(* Logix 5000 project; controller P1 vendor 1 type 14 code 92 rev 20.55; software revision 20.01 *)

TASK MainTask (continuous, watchdog 500 ms) : MainProgram

MODULES
   Local : vendor 1 type 14 code 92 (ICP 0, rev 20.55)
      P1_EN2T_PCN : 1756-EN2T (ICP 1, Ethernet 192.168.1.10, rev 10.1)
         P6 : 1756-EN2T (Ethernet 192.168.1.60, rev 10.1, Output RPI 10 ms)
            P6_CONTROLLER : vendor 1 type 14 code 92 (ICP 0, rev 20.1)
         P2 : 1756-EN2T (Ethernet 192.168.1.20, rev 10.7, Output RPI 10 ms)
            P2_CONTROLLER : vendor 1 type 14 code 92 (ICP 0, rev 20.1)
         P5 : 1756-EN2T (Ethernet 192.168.1.50, rev 10.1, Output RPI 10 ms)
            P5_CONTROLLER : vendor 1 type 14 code 92 (ICP 0, rev 20.1)
         P3 : 1756-EN2T (Ethernet 192.168.1.30, rev 10.7, Output RPI 10 ms)
            P3_CONTROLLER : vendor 1 type 14 code 92 (ICP 0, rev 20.1)
         P4 : 1756-EN2T (Ethernet 192.168.1.40, rev 10.1, Output RPI 10 ms)
            P4_CONTROLLER : vendor 1 type 14 code 92 (ICP 0, rev 20.1)
      P1_EN2TR_RIO : vendor 1 type 12 code 200 (ICP 2, Ethernet 192.168.0.10, rev 10.1)
         RIO1 : 1794-AENTR (Ethernet 192.168.0.12, rev 1.1, Output RPI 20 ms)
            RIO1_DI : 1794-IB32 (Flex 0, rev 1.1, Input RPI 20 ms)
            RIO1_DO : vendor 1 type 7 code 35 (Flex 1, rev 1.1)
            RIO1_AI : 1794-IE12 (Flex 2, rev 1.1, Output RPI 80 ms)
         WRIO1 : vendor 309 type 12 code 1000 (Ethernet 192.168.0.15, rev 3.1, Output RPI 20 ms)
            WRIO1_AI : 1734-IE2C (PointIO 1, rev 3.1, Input RPI 80 ms)
END_MODULES

TYPE AIN_UDT :
STRUCT
   Pv : REAL;
   Heu : REAL;
   Leu : REAL;
   SAHH : REAL;
   SAH : REAL;
   SAL : REAL;
   SALL : REAL;
   AHH : BOOL;
   AH : BOOL;
   AL : BOOL;
   ALL : BOOL;
   Wifi_Enb : BOOL;
   Hty : BOOL;
   Sim : BOOL;
   Sim_PV : REAL;
END_STRUCT
END_TYPE

TYPE AUTOINP_UDT :
STRUCT
   ON : BOOL;
END_STRUCT
END_TYPE

TYPE ControllerLEDStatus :
STRUCT
   Off : BOOL;
   SolidGreen : BOOL;
   FlashingGreen : BOOL;
   SolidYellow : BOOL;
   FlashingYellow : BOOL;
   FlashingRed : BOOL;
   SolidRed : BOOL;
END_STRUCT
END_TYPE

TYPE Duty2_UDT :
STRUCT
   Selection : INT;
   Pump_Running : BOOL;
   Selected_Pmp_Not_Avl : BOOL;
   Both_Pmp_Not_Avl : BOOL;
END_STRUCT
END_TYPE

TYPE FaultRecord :
STRUCT
   timelow : DINT;
   timehigh : DINT;
   type : INT;
   code : INT;
   info : DINT[8];
END_STRUCT
END_TYPE

TYPE FIT_UDT :
STRUCT
   Pv : REAL;
   Heu : REAL;
   Leu : REAL;
   SAHH : REAL;
   SAH : REAL;
   SAL : REAL;
   SALL : REAL;
   Totaliser : REAL;
   AHH : BOOL;
   AH : BOOL;
   AL : BOOL;
   ALL : BOOL;
   Sim : BOOL;
   Sim_PV : REAL;
   Wifi_Enb : BOOL;
   Rst_Totaliser : BOOL;
   Hty : BOOL;
END_STRUCT
END_TYPE

TYPE Logix_Status_FP :
STRUCT
   ClearMinorFaults : DINT;
   Sts_MinorFaultEvents : DINT;
   Sts_MinorFaultBits : DINT;
   Sts_Redundant : DINT;
   Set_FaceplateAnimation : DINT;
   Val_ProductCode : DINT;
   MemoryTemp : INT[29];
   Val_raw_data : INT;
   Sts_IO_LED_raw : INT;
   Sts_ProductCode : INT;
   Val_Force_data_raw : INT;
   MemoryRequestData : SINT[12];
   Sts_Force_Installed : BOOL;
   Sts_Force_Enabled : BOOL;
   Sts_Faulted : BOOL;
   Sts_Run : BOOL;
   Sts_Program : BOOL;
   Sts_Minor_fault : BOOL;
   Sts_Major_fault : BOOL;
   Sts_KS_in_run : BOOL;
   Sts_KS_in_program : BOOL;
   Sts_KS_in_remote : BOOL;
   Sts_Changingmodes : BOOL;
   Sts_Test : BOOL;
   Sts_Ladder_Working : BOOL;
   Cmd_ClearFaultRecord : BOOL;
   Set_Controller_Description : STRING;
   UpdateDelayTimer : TIMER;
   Val_MajorFault : FaultRecord;
   Val_MFS : FaultRecord;
   Sts_IO_LED : ControllerLEDStatus;
   Sts_Battery_LED : ControllerLEDStatus;
   MemoryData : Memory_Data;
   TEST : DINT;
END_STRUCT
END_TYPE

TYPE Memory_Data :
STRUCT
   Free_Mem_IO : DINT;
   Free_Mem_DT : DINT;
   Free_Memory : DINT;
   Total_Mem_IO : DINT;
   Total_Mem_DT : DINT;
   Total_Memory : DINT;
   Biggest_IO_Mem_Size_Ava : DINT;
   Biggest_DT_Mem_Size_Ava : DINT;
END_STRUCT
END_TYPE

TYPE MV_UDT :
STRUCT
   Cmd : INT;
   Status : INT;
   Reset : BOOL;
   Auto : BOOL;
   FTO : BOOL;
   FTC : BOOL;
   Avl : BOOL;
END_STRUCT
END_TYPE

TYPE PLANT_AUTO_UDT :
STRUCT
   ON : BOOL;
   OFF : BOOL;
END_STRUCT
END_TYPE

TYPE PLANT_UDT :
STRUCT
   START : BOOL;
   STOP : BOOL;
END_STRUCT
END_TYPE

TYPE PMP_UDT :
STRUCT
   Cmd : INT;
   Status : INT;
   RunMin : REAL;
   Total_RunMin : REAL;
   RunHr : REAL;
   Total_RunHr : REAL;
   Remote : BOOL;
   Auto : BOOL;
   Fault : BOOL;
   Avl : BOOL;
   Permissive : DINT;
   Shutdown : DINT;
   SD : DINT;
   Reset : BOOL;
   Reset_RunHr : BOOL;
   FTR : BOOL;
   FTS : BOOL;
END_STRUCT
END_TYPE

TYPE PRECONDITION_UDT :
STRUCT
   PERMISSIVE1 : BOOL;
   PERMISSIVE2 : BOOL;
   PERMISSIVE3 : BOOL;
   PERMISSIVE4 : BOOL;
   PERMISSIVE5 : BOOL;
   SHUTODWN1 : BOOL;
   SHUTODWN2 : BOOL;
   SHUTODWN3 : BOOL;
   SHUTODWN4 : BOOL;
   SHUTODWN5 : BOOL;
END_STRUCT
END_TYPE

TYPE RED_STAT :
STRUCT
   Redundancy_status_of_the_controller : INT;
   Redundancy_state_of_the_partner : INT;
END_STRUCT
END_TYPE

TYPE WIFI_UDT :
STRUCT
   PLC_WIFI : BOOL;
   RIO_WIFI : BOOL;
END_STRUCT
END_TYPE

ADD_ON_INSTRUCTION AIN_FBD   (* revision 1.0 *)
VAR_INPUT
   WRIO_Enb : BOOL; {visible}
   Raw_RIO : INT; {visible}
   Raw_WRIO : INT; {visible}
   L_Raw_RIO : INT; {visible}
   H_Raw_RIO : INT; {visible}
   L_Raw_WRIO : INT; {visible}
   H_Raw_WRIO : INT; {visible}
   HEU : INT; {visible}
   LEU : INT; {visible}
END_VAR
VAR_OUTPUT
   Hty : BOOL; {visible}
   Wifi_Enb : BOOL; {access Read Only, visible}
   AHH : BOOL; {visible}
   AH : BOOL; {access Read Only, visible}
   AL : BOOL; {access Read Only, visible}
   ALL : BOOL; {visible}
END_VAR
VAR_INPUT
   SAHH : REAL; {visible}
   SAH : REAL; {visible}
   SAL : REAL; {visible}
   SALL : REAL; {visible}
   Simulation : BOOL; {visible}
   RIO_Hty : BOOL; {visible}
   WRIO_Hty : BOOL; {visible}
END_VAR
VAR_IN_OUT
   Pv : REAL; {required}
   Sim_PV : REAL; {required}
   HMI : AIN_UDT; {required}
END_VAR
VAR
   SCALE : SCALE; {access None}
   ALM : ALARM; {access None}
   _Raw : INT; {access None}
   _L_Raw : INT; {access None}
   _H_Raw : INT; {access None}
   _Inst_Hty : BOOL; {access None}
END_VAR

ROUTINE Logic   (* structured text *)
   (*RIO and Wireless RIO Selection*)
   
   IF WRIO_Enb THEN
   	Wifi_Enb	:= 1;
   	_Raw		:= Raw_WRIO;
   	_H_Raw		:= H_Raw_WRIO;
   	_L_Raw		:= L_Raw_WRIO;
   	_Inst_Hty 	:= WRIO_Hty;
   ELSE
   	Wifi_Enb	:= 0;
   	_Raw		:= Raw_RIO;
   	_H_Raw		:= H_Raw_RIO;
   	_L_Raw		:= L_Raw_RIO;
   	_Inst_Hty 	:= RIO_Hty;
   END_IF;
   
   (*Calculation for PV*)
   IF Simulation THEN
   	Pv	:=Sim_PV;
   ELSE
   	SCALE.In		:=_Raw;
   	SCALE.InRawMax	:=_H_Raw;
   	SCALE.InRawMin	:=_L_Raw;
   	SCALE.InEUMax	:=HEU;
   	SCALE.InEUMin	:=LEU;
   	SCL(SCALE);
   
   	IF SCALE.Out<0 THEN
   		Pv	:= 0.0;
   	ELSE
   		Pv	:=SCALE.Out;
   	END_IF;
   
   	Sim_PV	:=Pv;
   
   END_IF;
   
   (*Alarms*)
   ALM.In			:=Pv;
   ALM.HHLimit		:=SAHH;
   ALM.HLimit		:=SAH;
   ALM.LLimit		:=SAL;
   ALM.LLLimit		:=SALL;
   ALM(ALM);
   
   AHH				:=ALM.HHAlarm;
   AH				:=ALM.HAlarm;
   AL				:=ALM.LAlarm;
   ALL				:=ALM.LLAlarm;
   
   Hty:= _Inst_Hty AND (_Raw > _L_Raw) AND (_Raw < _H_Raw)  ;
   
   
   
   
   
   
END_ROUTINE
END_ADD_ON_INSTRUCTION

ADD_ON_INSTRUCTION Duty2_FBD   (* revision 1.0 *)
VAR_INPUT
   AutoInp : BOOL; {visible}
   Selection : INT; {visible}
END_VAR
VAR_OUTPUT
   Start_Pmp1 : BOOL; {visible}
   Start_Pmp2 : BOOL; {visible}
END_VAR
VAR_IN_OUT
   PMP1 : PMP_UDT; {required}
   PMP2 : PMP_UDT; {required}
   HMI : Duty2_UDT; {required}
END_VAR

ROUTINE Logic   (* structured text *)
   IF PMP1.Status=2 OR PMP2.Status=2 THEN
   	HMI.Pump_Running := 1;
   ELSE
   	HMI.Pump_Running := 0;
   END_IF;
   
   HMI.Both_Pmp_Not_Avl		:= NOT PMP1.Avl AND NOT PMP2.Avl;
   
   IF AutoInp THEN
   	CASE Selection OF
   		(*PUMP 1 *)
   		1:
   			IF PMP1.Avl THEN
   				Start_Pmp1					:=1;
   				Start_Pmp2					:=0;
   				HMI.Selected_Pmp_Not_Avl	:=0;
   			ELSIF NOT PMP1.Avl AND PMP2.Avl THEN
   				Start_Pmp1					:=0;
   				Start_Pmp2					:=1;
   				HMI.Selected_Pmp_Not_Avl	:=1;
   			ELSIF NOT PMP1.Avl AND NOT PMP2.Avl	THEN
   				Start_Pmp1					:=0;
   				Start_Pmp2					:=0;
   			ELSE
   				HMI.Selected_Pmp_Not_Avl	:=0;
   			END_IF;
   
   		(*PUMP 2 *)
   		2:
   			IF PMP2.Avl THEN
   				Start_Pmp1					:=0;
   				Start_Pmp2					:=1;
   				HMI.Selected_Pmp_Not_Avl	:=0;
   			ELSIF NOT PMP2.Avl AND PMP1.Avl THEN
   				Start_Pmp1					:=1;
   				Start_Pmp2					:=0;
   				HMI.Selected_Pmp_Not_Avl	:=1;
   			ELSIF NOT PMP1.Avl AND NOT PMP2.Avl	THEN
   				Start_Pmp1					:=0;
   				Start_Pmp2					:=0;
   			ELSE
   				HMI.Selected_Pmp_Not_Avl	:=0;
   			END_IF;
   	END_CASE;
   ELSE
   	Start_Pmp1					:=0;
   	Start_Pmp2					:=0;
   END_IF;
   
   
END_ROUTINE
END_ADD_ON_INSTRUCTION

ADD_ON_INSTRUCTION FIT_FBD   (* revision 1.0 *)
VAR_INPUT
   WRIO_Enb : BOOL; {visible}
   Raw_RIO : INT; {visible}
   Raw_WRIO : INT; {visible}
   L_Raw_RIO : INT; {visible}
   H_Raw_RIO : INT; {visible}
   L_Raw_WRIO : INT; {visible}
   H_Raw_WRIO : INT; {visible}
   HEU : REAL; {visible}
   LEU : REAL; {visible}
END_VAR
VAR_OUTPUT
   Hty : BOOL; {visible}
   Wifi_Enb : BOOL; {visible}
   AHH : BOOL; {visible}
   AH : BOOL; {access Read Only, visible}
   AL : BOOL; {access Read Only, visible}
   ALL : BOOL; {visible}
END_VAR
VAR_INPUT
   SAHH : REAL; {visible}
   SAH : REAL; {visible}
   SAL : REAL; {visible}
   SALL : REAL; {visible}
   Simulation : BOOL; {visible}
   RIO_Hty : BOOL; {visible}
   WRIO_Hty : BOOL; {visible}
   Totaliser_Enb : BOOL; {visible}
   Rst_Totaliser : BOOL; {visible}
END_VAR
VAR_IN_OUT
   Totaliser : REAL; {required}
   Pv : REAL; {required}
   Sim_Pv : REAL; {required}
   HMI : FIT_UDT; {required}
END_VAR
VAR
   SCALE : SCALE; {access None}
   ALM : ALARM; {access None}
   TON : FBD_TIMER; {access None}
   _SEC_P : BOOL; {access None}
   _Inst_Hty : BOOL; {access None}
   _L_Raw : INT; {access None}
   _H_Raw : INT; {access None}
   _Raw : INT; {access None}
   R_TRIG : FBD_ONESHOT; {access None}
END_VAR

ROUTINE Logic   (* structured text *)
   (*RIO and Wireless RIO Selection*)
   
   IF WRIO_Enb THEN
   	Wifi_Enb	:= 1;
   	_Raw		:= Raw_WRIO;
   	_H_Raw		:= H_Raw_WRIO;
   	_L_Raw		:= L_Raw_WRIO;
   	_Inst_Hty 	:= WRIO_Hty;
   ELSE
   	Wifi_Enb	:= 0;
   	_Raw		:= Raw_RIO;
   	_H_Raw		:= H_Raw_RIO;
   	_L_Raw		:= L_Raw_RIO;
   	_Inst_Hty 	:= RIO_Hty;
   END_IF;
   
   (*Calculation for PV*)
   IF Simulation THEN
   	Pv	:= Sim_Pv   ;
   ELSE
   	SCALE.In		:=_Raw;
   	SCALE.InRawMax	:=_H_Raw;
   	SCALE.InRawMin	:=_L_Raw;
   	SCALE.InEUMax	:=HEU;
   	SCALE.InEUMin	:=LEU;
   	SCL(SCALE);
   	IF SCALE.Out>0 THEN
   		Pv	:=SCALE.Out;
   	ELSIF SCALE.Out<=0 THEN
   		Pv	:=0.0;
   	END_IF;
   
   	Sim_Pv	:=Pv;
   END_IF;
   
   (*Alarms*)
   ALM.In			:=Pv;
   ALM.HHLimit		:=SAHH;
   ALM.HLimit		:=SAH;
   ALM.LLimit		:=SAL;
   ALM.LLLimit		:=SALL;
   ALM(ALM);
   
   AHH				:=ALM.HHAlarm;
   AH				:=ALM.HAlarm;
   AL				:=ALM.LAlarm;
   ALL				:=ALM.LLAlarm;
   
   (*SECOND PULSE*)
   TON.PRE	:=1000;
   TON.TimerEnable	:=1;
   TONR(TON );
   R_TRIG.InputBit :=TON.DN ;
   OSRI( R_TRIG);
   _SEC_P  := R_TRIG.OutputBit;
   TON.Reset := _SEC_P;
   
   IF Totaliser_Enb THEN
   	IF _SEC_P THEN
   		HMI.Totaliser := HMI.Totaliser +  (ABS(Pv) / 3600 );
   	END_IF;
   END_IF;
   
   IF  Rst_Totaliser   THEN
   	HMI.Totaliser	:=0;
   END_IF;
   
   Hty:= _Inst_Hty AND (_Raw > _L_Raw) AND (_Raw < _H_Raw)  ;
   
   
   
   
   
   
END_ROUTINE
END_ADD_ON_INSTRUCTION

ADD_ON_INSTRUCTION MV_FBD   (* revision 1.0 *)
VAR_INPUT
   Auto : BOOL; {visible}
END_VAR
VAR_OUTPUT
   Cmd_Open : BOOL; {visible}
   Cmd_Close : BOOL; {visible}
   FTO : BOOL; {visible}
   FTC : BOOL; {access Read Only, visible}
END_VAR
VAR_INPUT
   AutoInp : BOOL; {visible}
   ZSO : BOOL; {visible}
   Open_TM : DINT; {visible}
   ZSC : BOOL; {visible}
   Close_TM : DINT; {visible}
END_VAR
VAR_IN_OUT
   Cmd : INT; {required}
   HMI : MV_UDT; {required}
END_VAR
VAR
   TON_Open_TM : FBD_TIMER; {access None}
   TON_Close_TM : FBD_TIMER; {access None}
END_VAR

ROUTINE Logic   (* structured text *)
   (*Fail to Close*)
   TON_Close_TM.PRE 			:= 	Close_TM*1000;
   TON_Close_TM.TimerEnable 	:=  Cmd_Close;
   TONR(TON_Close_TM);
   
   (*Fail to Open*)
   TON_Open_TM.PRE 			:= 	Open_TM*1000;
   TON_Open_TM.TimerEnable 	:= 	Cmd_Open;
   TONR(TON_Open_TM);
   
   IF ZSC THEN
   	HMI.Status	:=1;
   ELSIF ZSO THEN
   	HMI.Status	:=2;
   ELSE
   	HMI.Status	:=0;
   END_IF;
   
   HMI.Avl:= Auto AND NOT FTC AND NOT FTO;
   
   IF HMI.Reset THEN
   	(*IF NOT TON_Close_TM.DN AND ZSC THEN*)
   			FTC		:= 0;
   	(*END_IF;*)
   	(*IF NOT TON_Open_TM.DN AND ZSO THEN*)
   			FTO		:= 0;
   	(*END_IF;*)
   END_IF;
   
   IF  NOT Auto THEN
   	CASE HMI.Cmd OF
   		1:	(*CLOSE*)
   			Cmd_Close	:= 1;
   			Cmd_Open	:= 0;
   			IF TON_Close_TM.DN AND (NOT ZSC) THEN
   				FTC		:= 1;
   				FTO		:= 0;
   			END_IF;
   		2:	(*OPEN*)
   			IF FTO OR FTC    THEN
   				HMI.Cmd := 1;
   			END_IF;
   
   			IF NOT FTC AND NOT FTO THEN
   				Cmd_Close	:= 0;
   				Cmd_Open	:= 1;
   			END_IF;
   
   			IF TON_Open_TM.DN AND (NOT ZSO) THEN
   				FTC		:= 0;
   				FTO		:= 1;
   				HMI.Cmd := 1;
   			END_IF;
   	END_CASE;
   ELSE
   	(*Maintain Last status when switching from Auto to Manual*)
   	IF ZSO THEN
   		Cmd	:= 2;
   	END_IF;
   	IF ZSC THEN
   		Cmd	:= 1;
   	END_IF;
   
   	IF  AutoInp AND (NOT FTC AND NOT FTO) THEN
   		Cmd_Close	:= 0;
   		Cmd_Open	:= 1;
   		IF TON_Open_TM.DN AND (NOT ZSO) THEN
   			FTC		:= 0;
   			FTO		:= 1;
   		END_IF;
   	ELSE
   		Cmd_Close	:= 1;
   		Cmd_Open	:= 0;
   		IF TON_Close_TM.DN AND (NOT ZSC) THEN
   			FTC		:= 1;
   			FTO		:= 0;
   		END_IF;
   	END_IF;
   END_IF;
   
   
END_ROUTINE
END_ADD_ON_INSTRUCTION

ADD_ON_INSTRUCTION PMP_FBD   (* revision 1.0 *)
VAR_OUTPUT
   Cmd_Start : BOOL; {visible}
   Avl : BOOL; {visible}
   Fault : BOOL; {visible}
   FT_Stop : BOOL; {visible}
   FT_Start : BOOL; {visible}
   RunHr : REAL; {visible}
   Total_RunHr : REAL; {visible}
   SD : DINT; {access Read Only, visible}
END_VAR
VAR_INPUT
   Auto : BOOL; {visible}
   AutoInp : BOOL; {visible}
   Remote : BOOL; {visible}
   Run : BOOL; {visible}
   Trip : BOOL; {visible}
   Start_TM : DINT; {visible}
   Stop_TM : DINT; {visible}
   Rst : BOOL; {visible}
   Rst_RunHr : BOOL; {visible}
   Permissive : DINT; {visible}
   Shutdown : DINT; {visible}
END_VAR
VAR_IN_OUT
   RunMin : REAL; {required}
   Total_RunMin : REAL; {required}
   Cmd : INT; {required}
   HMI : PMP_UDT; {required}
END_VAR
VAR
   TON_Start_TM : FBD_TIMER; {access None}
   TON_Stop_TM : FBD_TIMER; {access None}
   _Min_P : BOOL; {access None}
   TON_Min : FBD_TIMER; {access None}
   R_TRIG_SEC : FBD_ONESHOT; {access None}
END_VAR

ROUTINE Logic   (* structured text *)
   (*Fail to Start*)
   TON_Start_TM.PRE 			:= 	Start_TM*1000;
   TON_Start_TM.TimerEnable 	:=  Cmd_Start;
   TONR(TON_Start_TM);
   
   (*Fail to Stop*)
   TON_Stop_TM.PRE 			:= 	Stop_TM*1000;
   TON_Stop_TM.TimerEnable 	:=  NOT Cmd_Start;
   TONR(TON_Stop_TM);
   
   IF (NOT Run) THEN
   	HMI.Status	:=1;
   ELSE
   	HMI.Status	:=2;
   END_IF;
   
   IF Fault THEN
   	HMI.Fault:= 1;
   ELSE
   	HMI.Fault:= 0;
   END_IF;
   
   IF HMI.Reset THEN
   	IF NOT TON_Stop_TM.DN THEN
   			FT_Stop		:= 0;
   	END_IF;
   	IF NOT TON_Start_TM.DN THEN
   			FT_Start	:= 0;
   	END_IF;
   
   	SD :=0;
   
   END_IF;
   
   Fault		:=Trip OR SD<>0;
   HMI.Remote	:=Remote;
   Avl:= Auto AND Remote AND NOT Fault AND NOT FT_Start AND NOT FT_Stop AND SD=0 ;
   
   IF Remote THEN
   	IF  NOT Auto THEN
   		CASE HMI.Cmd OF
   			1:	(*Stop*)
   				Cmd_Start	:=0;
   				IF TON_Stop_TM.DN AND Run THEN
   					FT_Start	:= 0;
   					FT_Stop		:= 1;
   				END_IF;
   			2:	(*OPEN*)
   				IF NOT Fault AND NOT FT_Start AND NOT FT_Stop AND (Permissive=-1) AND HMI.SD=0 THEN
   					Cmd_Start	:= 1;
   				ELSIF Cmd_Start AND (HMI.SD<>0) OR Fault THEN
   					SD				:= HMI.SD;
   					Cmd_Start		:= 0;
   					HMI.Cmd 		:= 1;
   				ELSIF (Permissive<>-1) THEN
   					HMI.Cmd 		:= 1;
   				END_IF;
   
   				IF TON_Start_TM.DN AND NOT Run THEN
   					FT_Start	:= 1;
   					FT_Stop		:= 0;
   					Cmd_Start	:= 0;
   					HMI.Cmd 	:= 1;
   				END_IF;
   		END_CASE;
   	ELSE
   		IF Run THEN
   			Cmd	:= 2;
   		END_IF;
   		IF (NOT Run) OR Fault OR FT_Start OR FT_Stop THEN
   			Cmd	:= 1;
   		END_IF;
   
   		IF  AutoInp  THEN
   			IF NOT Fault AND NOT FT_Start AND NOT FT_Stop AND (Permissive=-1) AND HMI.SD=0  THEN
   				Cmd_Start	:=1;
   			ELSIF Cmd_Start OR (HMI.SD<>0) OR Fault THEN
   				SD			:= HMI.SD;
   				Cmd_Start	:=0;
   			END_IF;
   
   			IF TON_Start_TM.DN AND NOT Run THEN
   				FT_Start	:= 1;
   				FT_Stop		:= 0;
   				Cmd_Start	:= 0;
   				HMI.Cmd 	:= 1;
   			END_IF;
   		ELSE
   			Cmd_Start	:=0;
   			IF TON_Stop_TM.DN AND Run THEN
   				FT_Start	:= 0;
   				FT_Stop		:= 1;
   
   			END_IF;
   		END_IF;
   	END_IF;
   
   ELSE (*Local*)
   	Cmd_Start	:=0;
   	Cmd	:= 1;
   
   	FT_Start	:= 0;
   	FT_Stop		:= 0;
   
   
   
   
   	(*	IF Run THEN
   			Cmd	:= 2;
   		END_IF;
   		IF (NOT Run) OR Fault OR FT_Start OR FT_Stop THEN
   			Cmd	:= 1;
   		END_IF;
   		*)
   END_IF;
   
   (*1 MIN PULSE*)
   TON_Min.PRE	:=60000;
   TON_Min.TimerEnable	:=1;
   TONR(TON_Min );
   R_TRIG_SEC.InputBit :=TON_Min.DN ;
   OSRI( R_TRIG_SEC);
   _Min_P  := R_TRIG_SEC.OutputBit;
   TON_Min.Reset 	:= _Min_P;
   
   IF Run THEN
   	IF _Min_P THEN
   		RunMin 			:=RunMin + 1.0;
   		Total_RunMin	:=Total_RunMin + 1.0;
   	END_IF;
   END_IF;
   
   RunHr 				:=RunMin/60.0;
   Total_RunHr			:=Total_RunMin/60.0;
   
   IF  Rst_RunHr THEN
   	RunMin	:=0;
   END_IF;
   
   
   
END_ROUTINE
END_ADD_ON_INSTRUCTION

VAR_GLOBAL   (* controller tags *)
   _FIT101_Tot_Enb : BOOL;
   _MIN_P : BOOL;
   _MV101_AutoInp : BOOL;
   _MV201_AutoInp : INT;
   _P_RAW_WATER_DUTY_AutoInp : BOOL;
   _PMP101_AutoInp : BOOL;
   _PMP102_AutoInp : BOOL;
   _SEC_P : BOOL;
   ADD_CLOSED : REAL := 0.7850342;
   ADD_OPEN : REAL := 0.98132324;
   AI_FIT_101_FLOW : INT := -30;
   AI_FIT_101_FLOW_HTY : BOOL := 1;
   AI_LIT_101_LEVEL : INT := 20823;
   AI_LIT_101_LEVEL_HTY : BOOL := 1;
   AI_RIO1_SPARE_03 : INT := -7700;
   AI_RIO1_SPARE_03_HTY : BOOL := 1;
   AI_RIO1_SPARE_04 : INT := -7701;
   AI_RIO1_SPARE_04_HTY : BOOL := 1;
   AI_RIO1_SPARE_05 : INT := -7702;
   AI_RIO1_SPARE_05_HTY : BOOL := 1;
   AI_RIO1_SPARE_06 : INT := -7702;
   AI_RIO1_SPARE_06_HTY : BOOL := 1;
   AI_RIO1_SPARE_07 : INT := -7704;
   AI_RIO1_SPARE_07_HTY : BOOL := 1;
   AI_RIO1_SPARE_08 : INT := -7701;
   AI_RIO1_SPARE_08_HTY : BOOL := 1;
   AI_RIO1_SPARE_09 : INT := -7702;
   AI_RIO1_SPARE_09_HTY : BOOL := 1;
   AI_RIO1_SPARE_10 : INT := -7704;
   AI_RIO1_SPARE_10_HTY : BOOL := 1;
   AI_RIO1_SPARE_11 : INT := -7700;
   AI_RIO1_SPARE_11_HTY : BOOL := 1;
   avg : REAL := 0.6411235;
   AVG_CLOSED : REAL := 0.13083903;
   AVG_OPEN : REAL := 0.16355388;
   DI_MV_101_ZSC : BOOL := 1;
   DI_MV_101_ZSO : BOOL;
   DI_P_101_AUTO : BOOL := 1;
   DI_P_101_FAULT : BOOL;
   DI_P_101_RUN : BOOL;
   DI_P_102_AUTO : BOOL;
   DI_P_102_FAULT : BOOL;
   DI_P_102_RUN : BOOL;
   DI_RIO1_SPARE_10 : BOOL;
   DI_RIO1_SPARE_11 : BOOL;
   DI_RIO1_SPARE_12 : BOOL;
   DI_RIO1_SPARE_13 : BOOL;
   DI_RIO1_SPARE_14 : BOOL;
   DI_RIO1_SPARE_15 : BOOL;
   DI_RIO1_SPARE_16 : BOOL;
   DI_RIO1_SPARE_17 : BOOL;
   DI_RIO1_SPARE_18 : BOOL;
   DI_RIO1_SPARE_19 : BOOL;
   DI_RIO1_SPARE_20 : BOOL;
   DI_RIO1_SPARE_21 : BOOL;
   DI_RIO1_SPARE_22 : BOOL;
   DI_RIO1_SPARE_23 : BOOL;
   DI_RIO1_SPARE_24 : BOOL;
   DI_RIO1_SPARE_25 : BOOL;
   DI_RIO1_SPARE_26 : BOOL;
   DI_RIO1_SPARE_27 : BOOL;
   DI_RIO1_SPARE_28 : BOOL;
   DI_RIO1_SPARE_29 : BOOL;
   DI_RIO1_SPARE_30 : BOOL;
   DI_RIO1_SPARE_31 : BOOL;
   DI_WIFI_PLC_1 : BOOL;
   DI_WIFI_RIO_1 : BOOL;
   DO_LED_RED : BOOL;
   DO_LED_RED1 : BOOL;
   DO_MV_101_CLOSE : BOOL := 1;
   DO_MV_101_OPEN : BOOL;
   DO_P_101_START : BOOL;
   DO_P_102_START : BOOL;
   DO_RIO1_SPARE_04 : BOOL;
   DO_RIO1_SPARE_05 : BOOL;
   DO_RIO1_SPARE_06 : BOOL;
   DO_RIO1_SPARE_07 : BOOL;
   DO_RIO1_SPARE_08 : BOOL;
   DO_RIO1_SPARE_09 : BOOL;
   DO_RIO1_SPARE_10 : BOOL;
   DO_RIO1_SPARE_11 : BOOL;
   DO_RIO1_SPARE_12 : BOOL;
   DO_RIO1_SPARE_13 : BOOL;
   DO_RIO1_SPARE_14 : BOOL;
   DO_RIO1_SPARE_15 : BOOL;
   dummy : BOOL; {access Read Only}
   dummy2 : BOOL := 1; {access Read Only}
   dummy_int : DINT := '$00$00$00$1E';
   Error_list_closed : REAL[20] := ([1] := 0.07849121, [3] := 0.07849121, [4] := 0.35327148, [5] := 0.27478027, [6] := 0.94207764, [7] := 0.7850342, [8] := 1.3345947, [9] := 1.4523315, [10] := 0.15704346);
   Error_list_open : REAL[20] := ([1] := 0.07849121, [2] := 0.07849121, [4] := 0.54956055, [5] := 0.27478027, [6] := 0.94207764, [7] := 0.7850342, [8] := 1.3345947, [9] := 1.4523315, [10] := 0.15704346);
   ERROR_P1_Ls : REAL := 0.07849121;
   first : BOOL := 1;
   FIT101_FB : FIT_FBD := (Raw_RIO := -30, Raw_WRIO := 3265, L_Raw_RIO := -15, H_Raw_RIO := 31208, L_Raw_WRIO := 3277, H_Raw_WRIO := 16383, HEU := 10.0, AL := 1, ALL := 1, SAHH := 4.0, SAH := 3.0, SAL := 1.0, SALL := 0.5, RIO_Hty := 1, WRIO_Hty := 1);
   HMI_FIT101 : FIT_UDT := (SAHH := 4.0, SAH := 3.0, SAL := 1.0, SALL := 0.5, Totaliser := 188.87244, AL := 1, ALL := 1);
   HMI_FIT102 : FIT_UDT;
   HMI_FIT201 : FIT_UDT := (SAHH := 3.5, SAH := 2.0, SALL := 0.4, Totaliser := 535.604, AL := 1, ALL := 1);
   HMI_FIT301 : FIT_UDT := (Pv := 0.0005124427, SAHH := 3.5, SAH := 3.0, Totaliser := 440.07816, Sim_PV := 0.0005124427, Hty := 1);
   HMI_LIT101 : AIN_UDT := (Pv := 817.2817, SAHH := 1000.0, SAH := 800.0, SAL := 500.0, SALL := 250.0, AH := 1, Hty := 1, Sim_PV := 817.2817);
   HMI_LIT301 : AIN_UDT := (Pv := 1008.3552, SAHH := 1200.0, SAH := 1000.0, SAL := 800.0, SALL := 250.0, AH := 1, Hty := 1, Sim_PV := 1008.3552);
   HMI_MV101 : MV_UDT := (Cmd := 1, Status := 1, Reset := 1, Auto := 1, Avl := 1);
   HMI_MV201 : MV_UDT := (Cmd := 1, Status := 1, Reset := 1, Auto := 1, Avl := 1);
   HMI_P101 : PMP_UDT := (Cmd := 1, Status := 1, RunMin := 831.0, Total_RunMin := 6892.0, RunHr := 13.85, Total_RunHr := 114.86667, Remote := 1, Auto := 1, Avl := 1, Permissive := -3, Reset := 1);
   HMI_P101_MSG : PRECONDITION_UDT := (PERMISSIVE1 := 1);
   HMI_P102 : PMP_UDT := (Cmd := 1, Status := 1, RunMin := 788.0, Total_RunMin := 788.0, RunHr := 13.133333, Total_RunHr := 13.133333, Auto := 1, Permissive := -3, Reset := 1);
   HMI_P102_MSG : PRECONDITION_UDT := (PERMISSIVE1 := 1);
   HMI_P1_PERMISSIVE : AUTOINP_UDT := (ON := 1);
   HMI_P1_READY : BOOL;
   HMI_P1_SHUTDOWN : BOOL := 1;
   HMI_P1_STATE : INT := 1;
   HMI_P2_PERMISSIVE : AUTOINP_UDT := (ON := 1);
   HMI_P3_PERMISSIVE : AUTOINP_UDT := (ON := 1);
   HMI_P4_PERMISSIVE : AUTOINP_UDT := (ON := 1);
   HMI_P5_PERMISSIVE : AUTOINP_UDT := (ON := 1);
   HMI_P5_SD_FLUSHING : AUTOINP_UDT;
   HMI_P5_SD_FLUSHING_DONE : AUTOINP_UDT;
   HMI_P5_STATE : INT := 1;
   HMI_P6_PERMISSIVE : AUTOINP_UDT := (ON := 1);
   HMI_P_RAW_WATER_DUTY : Duty2_UDT := (Selection := 1);
   HMI_PLANT : PLANT_UDT;
   HMI_PLANT_AUTO : PLANT_AUTO_UDT;
   HMI_PLANT_MANUAL : PLANT_AUTO_UDT;
   HMI_PLANT_READY : BOOL := 1;
   HMI_PLANT_RESET : PLANT_AUTO_UDT;
   HMI_SHUTDOWN_FLUSHING : AUTOINP_UDT;
   HMI_SHUTDOWN_TIMER : DINT := 13;
   HMI_START_PLANT : INT;
   HMI_STOP_PLANT : INT;
   HMI_WIFI : WIFI_UDT;
   LIT101_FB : AIN_FBD := (Raw_RIO := 20822, Raw_WRIO := 8736, H_Raw_RIO := 31208, L_Raw_WRIO := 3277, H_Raw_WRIO := 16383, HEU := 1225, Hty := 1, AH := 1, SAHH := 1000.0, SAH := 800.0, SAL := 500.0, SALL := 250.0, RIO_Hty := 1, WRIO_Hty := 1);
   LIT101_H_STATE : DINT := 5;
   LIT101_L_STATE : DINT;
   LIT101_LL_STATE : DINT;
   LIT301_H_STATE : DINT := 2;
   LIT301_L_STATE : DINT;
   LIT_101_Ls_PRV : REAL := 817.04614;
   LIT_101_MODEL_closed : REAL := 817.12463;
   LIT_101_MODEL_Ls : REAL := 813.1994;
   LIT_101_MODEL_Open : REAL := 817.04614;
   LIT_101_MODEL_PRV : REAL := 817.04614;
   LIT_STATE : DINT := 1;
   Logix_Status : Logix_Status_FP := (Set_FaceplateAnimation := 90, Val_ProductCode := 92, MemoryTemp[0] := 5, MemoryTemp[1] := 1, MemoryTemp[3] := 22852, MemoryTemp[4] := 3, MemoryTemp[5] := 7412, MemoryTemp[6] := 7, MemoryTemp[9] := 2, MemoryTemp[11] := -4608, MemoryTemp[12] := 3, MemoryTemp[14] := 8, MemoryTemp[17] := 5, MemoryTemp[21] := 6, MemoryTemp[23] := 20382, MemoryTemp[24] := 3, MemoryTemp[25] := 7, MemoryTemp[27] := 7372, MemoryTemp[28] := 7, Val_raw_data := 12640, Sts_IO_LED_raw := 2, Sts_ProductCode := 92, MemoryRequestData[0] := 5, MemoryRequestData[2] := 1, MemoryRequestData[4] := 2, MemoryRequestData[6] := 5, MemoryRequestData[8] := 6, MemoryRequestData[10] := 7, Sts_Run := 1, Sts_KS_in_remote := 1, Sts_Ladder_Working := 1, Set_Controller_Description := 'P1: Raw Water System', UpdateDelayTimer.PRE := 1000, UpdateDelayTimer.ACC := 990, UpdateDelayTimer.EN := 1, UpdateDelayTimer.TT := 1, Val_MFS.timelow := 71751885, Val_MFS.timehigh := 206334, Val_MFS.type := 3, Val_MFS.code := 20, Val_MFS.info[1] := 1, Sts_IO_LED.FlashingGreen := 1, Sts_Battery_LED.Off := 1, MemoryData.Free_Mem_IO := 877840, MemoryData.Free_Mem_DT := 1864656, MemoryData.Total_Mem_IO := 1030144, MemoryData.Total_Mem_DT := 2097152, MemoryData.Biggest_IO_Mem_Size_Ava := 867960, MemoryData.Biggest_DT_Mem_Size_Ava := 1864496);
   Memory_Message : MESSAGE;
        MessageParameters(ServiceCode := 16#0003, LocalElement := Logix_Status.MemoryRequestData[0], DestinationTag := Logix_Status.MemoryTemp[0], ...)
   MIN_TEST : DINT := 286354;
   MV101_FB : MV_FBD := (Auto := 1, Cmd_Close := 1, Open_TM := 15, ZSC := 1, Close_TM := 15);
   MV101_STATE : DINT := 6;
   n : DINT := 6;
   P101_FB : PMP_FBD := (Avl := 1, RunHr := 13.85, Total_RunHr := 114.86667, Auto := 1, Remote := 1, Start_TM := 3, Stop_TM := 3, Rst := 1, Permissive := -3);
   P101_STATE : DINT := 4;
   P102_FB : PMP_FBD := (RunHr := 13.133333, Total_RunHr := 13.133333, Auto := 1, Start_TM := 3, Stop_TM := 3, Rst := 1, Permissive := -3);
   P1_Status : INT;
   P2_AUTO_MSG : MESSAGE;
        MessageParameters(ServiceCode := 16#004d, LocalElement := HMI_PLANT_AUTO, ...)
   P2_FIT102_MSG : MESSAGE;
        MessageParameters(ServiceCode := 16#004c, LocalElement := HMI_FIT201, ...)
   P2_MV201_MSG : MESSAGE;
        MessageParameters(ServiceCode := 16#004c, LocalElement := HMI_MV201, ...)
   P2_PERM_MSG : MESSAGE;
        MessageParameters(ServiceCode := 16#004c, LocalElement := HMI_P2_PERMISSIVE, ...)
   P2_PLANT_MSG : MESSAGE;
        MessageParameters(ServiceCode := 16#004d, LocalElement := HMI_PLANT, ...)
   P2_RESET_MSG : MESSAGE;
        MessageParameters(ServiceCode := 16#004d, LocalElement := HMI_PLANT_RESET, ...)
   P2_SEND_MSG : MESSAGE;
        MessageParameters(ServiceCode := 16#004d, LocalElement := _MV201_AutoInp, ...)
   P3_AUTO_MSG : MESSAGE;
        MessageParameters(ServiceCode := 16#004d, LocalElement := HMI_PLANT_AUTO, ...)
   P3_FIT301_MSG : MESSAGE;
        MessageParameters(ServiceCode := 16#004c, LocalElement := HMI_FIT301, ...)
   P3_LIT301_MSG : MESSAGE;
        MessageParameters(ServiceCode := 16#004c, LocalElement := HMI_LIT301, ...)
   P3_PERM_MSG : MESSAGE;
        MessageParameters(ServiceCode := 16#004c, LocalElement := HMI_P3_PERMISSIVE, ...)
   P3_PLANT_MSG : MESSAGE;
        MessageParameters(ServiceCode := 16#004d, LocalElement := HMI_PLANT, ...)
   P3_RESET_MSG : MESSAGE;
        MessageParameters(ServiceCode := 16#004d, LocalElement := HMI_PLANT_RESET, ...)
   P4_AUTO_MSG : MESSAGE;
        MessageParameters(ServiceCode := 16#004d, LocalElement := HMI_PLANT_AUTO, ...)
   P4_PERM_MSG : MESSAGE;
        MessageParameters(ServiceCode := 16#004c, LocalElement := HMI_P4_PERMISSIVE, ...)
   P4_PLANT_MSG : MESSAGE;
        MessageParameters(ServiceCode := 16#004d, LocalElement := HMI_PLANT, ...)
   P4_RESET_MSG : MESSAGE;
        MessageParameters(ServiceCode := 16#004d, LocalElement := HMI_PLANT_RESET, ...)
   P5_AUTO_MSG : MESSAGE;
        MessageParameters(ServiceCode := 16#004d, LocalElement := HMI_PLANT_AUTO, ...)
   P5_PERM_MSG : MESSAGE;
        MessageParameters(ServiceCode := 16#004c, LocalElement := HMI_P5_PERMISSIVE, ...)
   P5_PLANT_MSG : MESSAGE;
        MessageParameters(ServiceCode := 16#004d, LocalElement := HMI_PLANT, ...)
   P5_PLANT_MSG_X : DINT;
   P5_RESET_MSG : MESSAGE;
        MessageParameters(ServiceCode := 16#004d, LocalElement := HMI_PLANT_RESET, ...)
   P5_SD_FLUSH_MSG : MESSAGE;
        MessageParameters(ServiceCode := 16#004c, LocalElement := HMI_P5_SD_FLUSHING_DONE, ...)
   P5_SD_FLUSHING_MSG : MESSAGE;
        MessageParameters(ServiceCode := 16#004d, LocalElement := HMI_SHUTDOWN_FLUSHING, ...)
   P5_STATE_MSG : MESSAGE;
        MessageParameters(ServiceCode := 16#004c, LocalElement := HMI_P5_STATE, ...)
   P6_AUTO_MSG : MESSAGE;
        MessageParameters(ServiceCode := 16#004d, LocalElement := HMI_PLANT_AUTO, ...)
   P6_PERM_MSG : MESSAGE;
        MessageParameters(ServiceCode := 16#004c, LocalElement := HMI_P6_PERMISSIVE, ...)
   P6_PLANT_MSG : MESSAGE;
        MessageParameters(ServiceCode := 16#004d, LocalElement := HMI_PLANT, ...)
   P6_RESET_MSG : MESSAGE;
        MessageParameters(ServiceCode := 16#004d, LocalElement := HMI_PLANT_RESET, ...)
   P_RAW_WATER_DUTY_FB : Duty2_FBD := (Selection := 1);
   ProtectTimer_SEC : INT;
   R_TRIG : FBD_ONESHOT;
   REDUNDANT_STATUS : RED_STAT := (Redundancy_status_of_the_controller := 2, Redundancy_state_of_the_partner := 8);
   RTRIG_MIN : FBD_ONESHOT;
   RTRIG_SEC : FBD_ONESHOT;
   SEC_COUNT : DINT := 1;
   SEC_TEST : INT;
   TEST_START : BOOL := 1;
   Threshold : REAL := 5.5;
   TON : FBD_TIMER;
   TON_FIT102_P1_TM : FBD_TIMER := (PRE := 10000);
   TON_FIT102_P2_TM : FBD_TIMER := (PRE := 10000);
   TON_FIT102_TM : FBD_TIMER := (PRE := 3000);
   TON_FIT201 : FBD_TIMER;
   TON_MIN : FBD_TIMER := (TimerEnable := 1, PRE := 60000, ACC := 57573, EN := 1, TT := 1);
   TON_SEC : FBD_TIMER := (TimerEnable := 1, PRE := 1000, ACC := 228, EN := 1, TT := 1);
   W_AI_FIT_101_FLOW : INT := 3265;
   W_AI_FIT_101_FLOW_HTY : BOOL := 1;
   W_AI_LIT_101_LEVEL : INT := 8736;
   W_AI_LIT_101_LEVEL_HTY : BOOL := 1;
END_VAR

PROGRAM MainProgram   (* main routine MainRoutine *)
VAR
   _MV_101_SR : DOMINANT_SET := (Reset := 1, OutNot := 1);
   _MV_201_SR : DOMINANT_SET;
   _P_RAW_WATER_DUTY_SR : DOMINANT_SET := (Reset := 1, OutNot := 1);
   ADD_CLOSED3 : REAL := 0.0021972656;
   ADD_OPEN3 : REAL := 0.0076904297;
   AVG_CLOSED3 : REAL := 0.00036621094;
   AVG_OPEN3 : REAL := 0.0012817383;
   count : DINT := 4;
   count1 : DINT;
   count3 : DINT := 4;
   Current_LIT101Level : DINT;
   Error_list_closed3 : REAL[10] := ([0] := 0.00036621094, [1] := 0.00036621094, [2] := 0.00036621094, [3] := 0.00036621094, [4] := 0.00036621094, [5] := 0.00036621094);
   Error_list_open3 : REAL[10] := ([0] := 0.00036621094, [1] := 0.0007324219, [2] := 0.0010986328, [3] := 0.0014648438, [4] := 0.0018310547, [5] := 0.0021972656);
   ERROR_P1_Open : REAL;
   ERROR_P3_Ls : REAL := 0.00036621094;
   ERROR_P3_Open : REAL := 0.0014648438;
   first3 : BOOL := 1;
   HMI_PLANT_START : BOOL := 1;
   i : DINT := 6;
   i3 : DINT := 6;
   LIT_301_Ls_PRV : REAL := 1008.3552;
   LIT_301_MODEL_closed : REAL := 1008.35486;
   LIT_301_MODEL_Open : REAL := 1008.35376;
   LIT_301_MODEL_PRV : REAL := 1008.35376;
   LIT_STATE3 : DINT := 2;
   n3 : DINT := 6;
   Previous_LIT101Level : DINT := 587;
   Threshold3 : REAL := 4.8;
   TIME_STATE : DINT := 5;
   TimeCount : BOOL;
   TimeToOverflow : DINT := -1;
END_VAR

ROUTINE IO   (* structured text *)
   
   
   
   (*DIGITAL INPUTS*)
   DI_WIFI_PLC_1		:=RIO1:0:I.Data.0;
   DI_WIFI_RIO_1		:=RIO1:0:I.Data.1;
   DI_P_101_AUTO		:=RIO1:0:I.Data.2;
   DI_P_101_RUN		:=RIO1:0:I.Data.3;
   DI_P_101_FAULT		:=RIO1:0:I.Data.4;
   DI_P_102_AUTO		:=RIO1:0:I.Data.5;
   DI_P_102_RUN		:=RIO1:0:I.Data.6;
   DI_P_102_FAULT		:=RIO1:0:I.Data.7;
   DI_MV_101_ZSO		:=RIO1:0:I.Data.8;
   DI_MV_101_ZSC		:=RIO1:0:I.Data.9;
   DI_RIO1_SPARE_10	:=RIO1:0:I.Data.10;
   DI_RIO1_SPARE_11	:=RIO1:0:I.Data.11;
   DI_RIO1_SPARE_12	:=RIO1:0:I.Data.12;
   DI_RIO1_SPARE_13	:=RIO1:0:I.Data.13;
   DI_RIO1_SPARE_14	:=RIO1:0:I.Data.14;
   DI_RIO1_SPARE_15	:=RIO1:0:I.Data.15;
   DI_RIO1_SPARE_16	:=RIO1:0:I.Data.16;
   DI_RIO1_SPARE_17	:=RIO1:0:I.Data.17;
   DI_RIO1_SPARE_18	:=RIO1:0:I.Data.18;
   DI_RIO1_SPARE_19	:=RIO1:0:I.Data.19;
   DI_RIO1_SPARE_20	:=RIO1:0:I.Data.20;
   DI_RIO1_SPARE_21	:=RIO1:0:I.Data.21;
   DI_RIO1_SPARE_22	:=RIO1:0:I.Data.22;
   DI_RIO1_SPARE_23	:=RIO1:0:I.Data.23;
   DI_RIO1_SPARE_24	:=RIO1:0:I.Data.24;
   DI_RIO1_SPARE_25	:=RIO1:0:I.Data.25;
   DI_RIO1_SPARE_26	:=RIO1:0:I.Data.26;
   DI_RIO1_SPARE_27	:=RIO1:0:I.Data.27;
   DI_RIO1_SPARE_28	:=RIO1:0:I.Data.28;
   DI_RIO1_SPARE_29	:=RIO1:0:I.Data.29;
   DI_RIO1_SPARE_30	:=RIO1:0:I.Data.30;
   DI_RIO1_SPARE_31	:=RIO1:0:I.Data.31;
   
   (*DIGITAL OUTPUTS*)
   RIO1:1:O.0	:=DO_P_101_START;
   RIO1:1:O.1	:=DO_P_102_START;
   RIO1:1:O.2	:=DO_MV_101_OPEN;
   RIO1:1:O.3	:=DO_MV_101_CLOSE;
   RIO1:1:O.4	:=DO_RIO1_SPARE_04;
   RIO1:1:O.5	:=DO_RIO1_SPARE_05;
   RIO1:1:O.6	:=DO_RIO1_SPARE_06;
   RIO1:1:O.7	:=DO_RIO1_SPARE_07;
   RIO1:1:O.8	:=DO_LED_RED;
   RIO1:1:O.9	:=DO_RIO1_SPARE_09;
   RIO1:1:O.10	:=DO_RIO1_SPARE_10;
   RIO1:1:O.11	:=DO_RIO1_SPARE_11;
   RIO1:1:O.12	:=DO_RIO1_SPARE_12;
   RIO1:1:O.13	:=DO_RIO1_SPARE_13;
   RIO1:1:O.14	:=DO_RIO1_SPARE_14;
   RIO1:1:O.15	:=DO_RIO1_SPARE_15;
   
   (*ANALOG INPUTS*)
   AI_LIT_101_LEVEL	:=RIO1:2:I.Ch0Data;
   AI_FIT_101_FLOW		:=RIO1:2:I.Ch1Data;
   AI_RIO1_SPARE_03	:=RIO1:2:I.Ch3Data;
   AI_RIO1_SPARE_04	:=RIO1:2:I.Ch4Data;
   AI_RIO1_SPARE_05	:=RIO1:2:I.Ch5Data;
   AI_RIO1_SPARE_06	:=RIO1:2:I.Ch6Data;
   AI_RIO1_SPARE_07	:=RIO1:2:I.Ch7Data;
   AI_RIO1_SPARE_08	:=RIO1:2:I.Ch8Data;
   AI_RIO1_SPARE_09	:=RIO1:2:I.Ch9Data;
   AI_RIO1_SPARE_10	:=RIO1:2:I.Ch10Data;
   AI_RIO1_SPARE_11	:=RIO1:2:I.Ch11Data;
   
   AI_LIT_101_LEVEL_HTY	:=(NOT RIO1:2:I.GeneralFault);
   AI_FIT_101_FLOW_HTY		:=(NOT RIO1:2:I.GeneralFault);
   AI_RIO1_SPARE_03_HTY	:=(NOT RIO1:2:I.GeneralFault);
   AI_RIO1_SPARE_04_HTY	:=(NOT RIO1:2:I.GeneralFault);
   AI_RIO1_SPARE_05_HTY	:=(NOT RIO1:2:I.GeneralFault);
   AI_RIO1_SPARE_06_HTY	:=(NOT RIO1:2:I.GeneralFault);
   AI_RIO1_SPARE_07_HTY	:=(NOT RIO1:2:I.GeneralFault);
   AI_RIO1_SPARE_08_HTY	:=(NOT RIO1:2:I.GeneralFault);
   AI_RIO1_SPARE_09_HTY	:=(NOT RIO1:2:I.GeneralFault);
   AI_RIO1_SPARE_10_HTY	:=(NOT RIO1:2:I.GeneralFault);
   AI_RIO1_SPARE_11_HTY	:=(NOT RIO1:2:I.GeneralFault);
   
   (*WIRELESS ANALOG INPUTS*)
   W_AI_LIT_101_LEVEL		:=WRIO1:1:I.Ch0Data;
   W_AI_FIT_101_FLOW		:=WRIO1:1:I.Ch1Data;
   
   W_AI_LIT_101_LEVEL_HTY	:=(NOT WRIO1:1:I.Ch0Fault);
   W_AI_FIT_101_FLOW_HTY	:=(NOT WRIO1:1:I.Ch1Fault);
   
   (*Wireless Selction*)
   HMI_WIFI.PLC_WIFI		:= DI_WIFI_PLC_1;
   HMI_WIFI.RIO_WIFI		:= DI_WIFI_RIO_1;
   
   
   
END_ROUTINE

ROUTINE Logix_Status   (* ladder *)
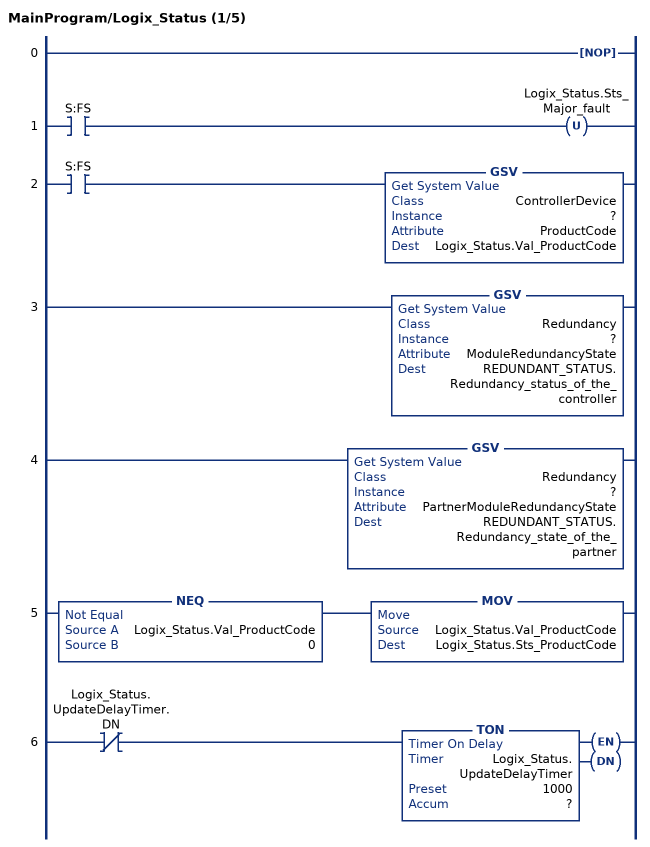
   0: NOP();
   1: XIC(S:FS)OTU(Logix_Status.Sts_Major_fault);
   2: XIC(S:FS)GSV(ControllerDevice,?,ProductCode,Logix_Status.Val_ProductCode);
   3: GSV(Redundancy,?,ModuleRedundancyState,REDUNDANT_STATUS.Redundancy_status_of_the_controller);
   4: GSV(Redundancy,?,PartnerModuleRedundancyState,REDUNDANT_STATUS.Redundancy_state_of_the_partner);
   5: NEQ(Logix_Status.Val_ProductCode,0)MOV(Logix_Status.Val_ProductCode,Logix_Status.Sts_ProductCode);
   6: XIO(Logix_Status.UpdateDelayTimer.DN)TON(Logix_Status.UpdateDelayTimer,?,?);
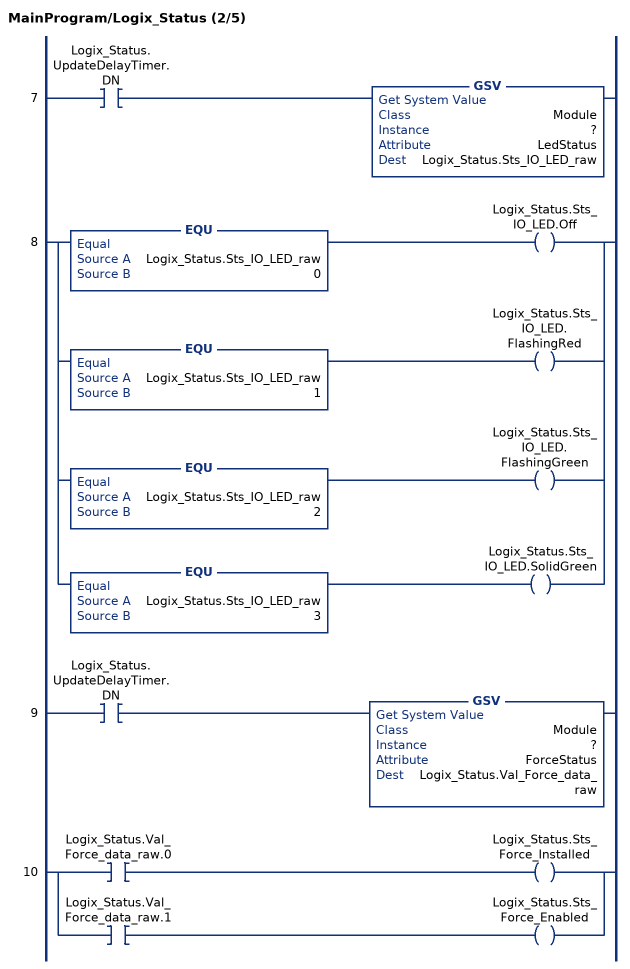
   7: XIC(Logix_Status.UpdateDelayTimer.DN)GSV(Module,?,LedStatus,Logix_Status.Sts_IO_LED_raw);
   8: [EQU(Logix_Status.Sts_IO_LED_raw,0) OTE(Logix_Status.Sts_IO_LED.Off) ,EQU(Logix_Status.Sts_IO_LED_raw,1) OTE(Logix_Status.Sts_IO_LED.FlashingRed) ,EQU(Logix_Status.Sts_IO_LED_raw,2) OTE(Logix_Status.Sts_IO_LED.FlashingGreen) ,EQU(Logix_Status.Sts_IO_LED_raw,3) OTE(Logix_Status.Sts_IO_LED.SolidGreen) ];
   9: XIC(Logix_Status.UpdateDelayTimer.DN)GSV(Module,?,ForceStatus,Logix_Status.Val_Force_data_raw);
   10: [XIC(Logix_Status.Val_Force_data_raw.0) OTE(Logix_Status.Sts_Force_Installed) ,XIC(Logix_Status.Val_Force_data_raw.1) OTE(Logix_Status.Sts_Force_Enabled) ];
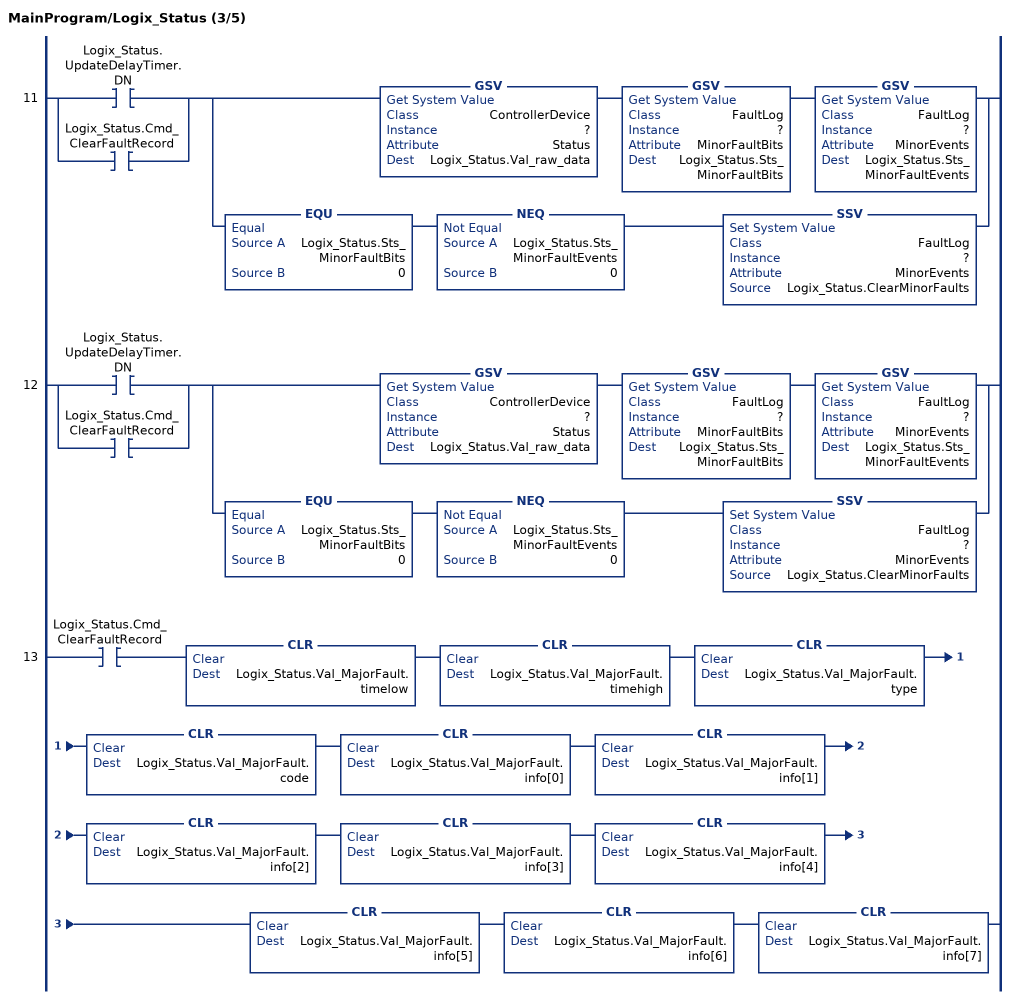
   11: [XIC(Logix_Status.UpdateDelayTimer.DN) ,XIC(Logix_Status.Cmd_ClearFaultRecord) ][GSV(ControllerDevice,?,Status,Logix_Status.Val_raw_data) GSV(FaultLog,?,MinorFaultBits,Logix_Status.Sts_MinorFaultBits) GSV(FaultLog,?,MinorEvents,Logix_Status.Sts_MinorFaultEvents) ,EQU(Logix_Status.Sts_MinorFaultBits,0) NEQ(Logix_Status.Sts_MinorFaultEvents,0) SSV(FaultLog,?,MinorEvents,Logix_Status.ClearMinorFaults) ];
   12: [XIC(Logix_Status.UpdateDelayTimer.DN) ,XIC(Logix_Status.Cmd_ClearFaultRecord) ][GSV(ControllerDevice,?,Status,Logix_Status.Val_raw_data) GSV(FaultLog,?,MinorFaultBits,Logix_Status.Sts_MinorFaultBits) GSV(FaultLog,?,MinorEvents,Logix_Status.Sts_MinorFaultEvents) ,EQU(Logix_Status.Sts_MinorFaultBits,0) NEQ(Logix_Status.Sts_MinorFaultEvents,0) SSV(FaultLog,?,MinorEvents,Logix_Status.ClearMinorFaults) ];
   13: XIC(Logix_Status.Cmd_ClearFaultRecord)CLR(Logix_Status.Val_MajorFault.timelow)CLR(Logix_Status.Val_MajorFault.timehigh)CLR(Logix_Status.Val_MajorFault.type)CLR(Logix_Status.Val_MajorFault.code)CLR(Logix_Status.Val_MajorFault.info[0])CLR(Logix_Status.Val_MajorFault.info[1])CLR(Logix_Status.Val_MajorFault.info[2])CLR(Logix_Status.Val_MajorFault.info[3])CLR(Logix_Status.Val_MajorFault.info[4])CLR(Logix_Status.Val_MajorFault.info[5])CLR(Logix_Status.Val_MajorFault.info[6])CLR(Logix_Status.Val_MajorFault.info[7]);
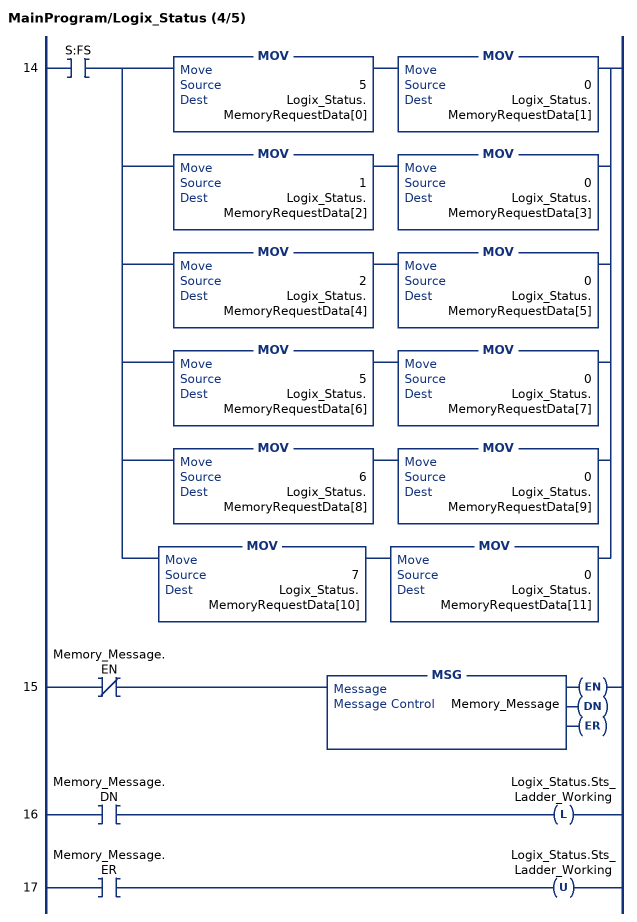
   14: XIC(S:FS)[MOV(5,Logix_Status.MemoryRequestData[0]) MOV(0,Logix_Status.MemoryRequestData[1]) ,MOV(1,Logix_Status.MemoryRequestData[2]) MOV(0,Logix_Status.MemoryRequestData[3]) ,MOV(2,Logix_Status.MemoryRequestData[4]) MOV(0,Logix_Status.MemoryRequestData[5]) ,MOV(5,Logix_Status.MemoryRequestData[6]) MOV(0,Logix_Status.MemoryRequestData[7]) ,MOV(6,Logix_Status.MemoryRequestData[8]) MOV(0,Logix_Status.MemoryRequestData[9]) ,MOV(7,Logix_Status.MemoryRequestData[10]) MOV(0,Logix_Status.MemoryRequestData[11]) ];
   15: XIO(Memory_Message.EN)MSG(Memory_Message);
   16: XIC(Memory_Message.DN)OTL(Logix_Status.Sts_Ladder_Working);
   17: XIC(Memory_Message.ER)OTU(Logix_Status.Sts_Ladder_Working);
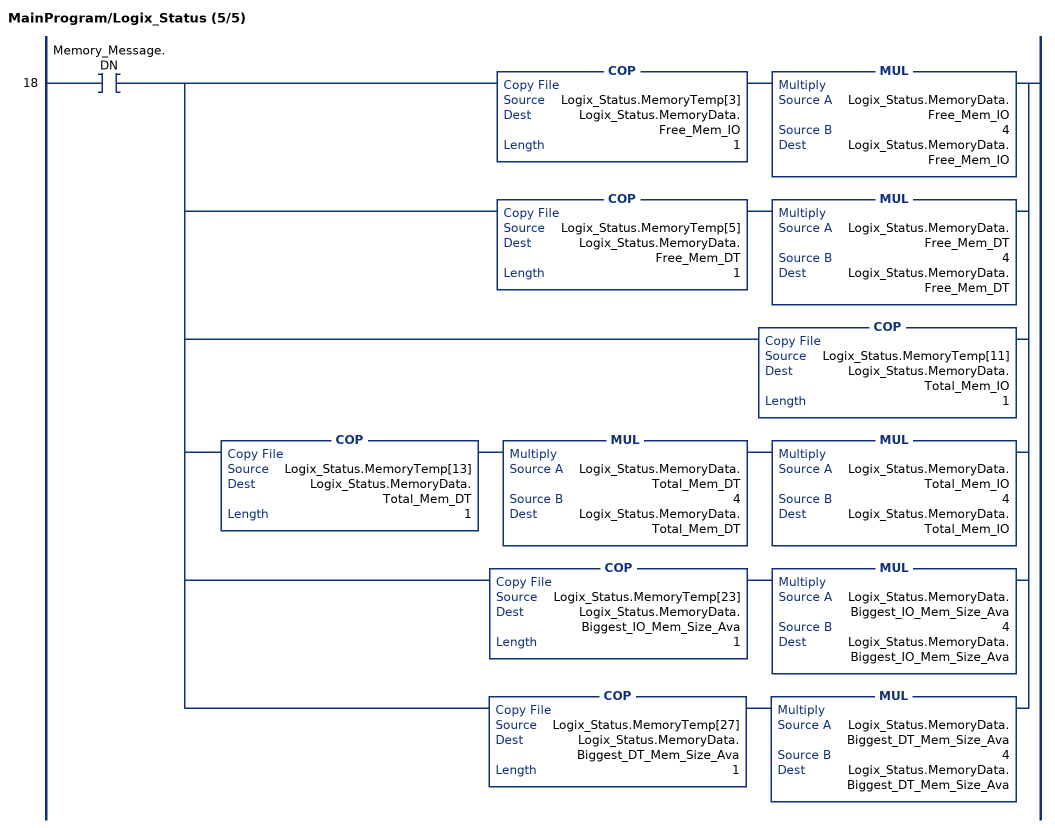
   18: XIC(Memory_Message.DN)[COP(Logix_Status.MemoryTemp[3],Logix_Status.MemoryData.Free_Mem_IO,1) MUL(Logix_Status.MemoryData.Free_Mem_IO,4,Logix_Status.MemoryData.Free_Mem_IO) ,COP(Logix_Status.MemoryTemp[5],Logix_Status.MemoryData.Free_Mem_DT,1) MUL(Logix_Status.MemoryData.Free_Mem_DT,4,Logix_Status.MemoryData.Free_Mem_DT) ,COP(Logix_Status.MemoryTemp[11],Logix_Status.MemoryData.Total_Mem_IO,1) ,COP(Logix_Status.MemoryTemp[13],Logix_Status.MemoryData.Total_Mem_DT,1) MUL(Logix_Status.MemoryData.Total_Mem_DT,4,Logix_Status.MemoryData.Total_Mem_DT) MUL(Logix_Status.MemoryData.Total_Mem_IO,4,Logix_Status.MemoryData.Total_Mem_IO) ,COP(Logix_Status.MemoryTemp[23],Logix_Status.MemoryData.Biggest_IO_Mem_Size_Ava,1) MUL(Logix_Status.MemoryData.Biggest_IO_Mem_Size_Ava,4,Logix_Status.MemoryData.Biggest_IO_Mem_Size_Ava) ,COP(Logix_Status.MemoryTemp[27],Logix_Status.MemoryData.Biggest_DT_Mem_Size_Ava,1) MUL(Logix_Status.MemoryData.Biggest_DT_Mem_Size_Ava,4,Logix_Status.MemoryData.Biggest_DT_Mem_Size_Ava) ];
END_ROUTINE

ROUTINE Main_Seq   (* structured text *)
   (*MINUTES PULSE*)
   TON_MIN.PRE	:=60000;
   TON_MIN.TimerEnable	:=1;
   TONR(TON_MIN );
   RTRIG_MIN.InputBit :=TON_MIN.DN ;
   OSRI( RTRIG_MIN);
   _MIN_P  := RTRIG_MIN.OutputBit;
   TON_MIN.Reset := _MIN_P;
   
   IF  _MIN_P      THEN
   	MIN_TEST:=MIN_TEST+1;
   
   END_IF;
   
   (*SECOND PULSE*)
   TON.PRE	:=1000;
   TON.TimerEnable	:=1;
   TONR(TON );
   R_TRIG.InputBit :=TON.DN ;
   OSRI( R_TRIG);
   _SEC_P  := R_TRIG.OutputBit;
   TON.Reset := _SEC_P;
   
   IF  _SEC_P      THEN
   	SEC_TEST:=SEC_TEST+1;
   
   END_IF;
   
   (*
   if S:FS then
   	HMI_P1_STATE := 1;
   end_if;
   *)
   
   
   
   
   (*
   IF HMI_P1_STATE =1 THEN
   	IF _MIN_P THEN
   		HMI_SHUTDOWN_TIMER:=HMI_SHUTDOWN_TIMER+1;
   	END_IF;
   
   	IF HMI_SHUTDOWN_TIMER>100  THEN
   		TEST_START:=1;
   		HMI_PLANT.START	:=1;
   			IF HMI_PLANT.START THEN
   				HMI_PLANT.START	:=0;
   			END_IF;
   
   		HMI_SHUTDOWN_FLUSHING.ON :=1;
   	ELSE
   		HMI_SHUTDOWN_FLUSHING.ON :=0;
   	END_IF;
   
   ELSE
   	HMI_SHUTDOWN_TIMER:=0;
   END_IF;
   *)
   
   IF HMI_PLANT.STOP THEN
   	HMI_P1_SHUTDOWN:=1;
   END_IF;
   
   
   //Passive Protection//
   //Water level increases by 125mm in 2 minutes//
   // When MV101 is set to Manual, and LIT101 is NOT in Simulation mode//
   IF HMI_LIT101.AHH THEN
   	IF _SEC_P THEN
   		ProtectTimer_SEC:=ProtectTimer_SEC+1;
   		IF ProtectTimer_SEC>120 THEN
   			HMI_MV101.Auto				:=1;
   			_MV101_AutoInp				:=0;
   		END_IF;
   	END_IF;
   END_IF;
   
   // When LIT101 is set to simulation mode, only allow 15 mins of Simulation Mode operation//
   IF HMI_LIT101.Sim THEN
   	IF _SEC_P THEN
   		ProtectTimer_SEC:=ProtectTimer_SEC+1;
   		IF ProtectTimer_SEC>900 THEN
   			HMI_LIT101.Sim 				:= 0;
   			IF HMI_LIT101.AHH or HMI_LIT101.AH THEN
   				HMI_MV101.Auto				:=1;
   				_MV101_AutoInp				:=0;
   			END_IF;
   		END_IF;
   	END_IF;
   END_IF;
   
   (*
   
   IF HMI_PLANT.STOP THEN
   	HMI_P1_STATE:=1;
   END_IF;
   *)
   
   (*-----------WRITE FAULT CONDITION--------------*)
   
   CASE HMI_P1_STATE OF
   	1:(*PLANT IN STANDBY*)
   		_MV101_AutoInp				:=0;
   		_P_RAW_WATER_DUTY_AutoInp	:=0;
   		HMI_P1_READY				:=0;
   
   		IF HMI_PLANT_READY AND HMI_PLANT.START AND HMI_P1_PERMISSIVE.ON  THEN
   			HMI_P1_STATE:=2;
   		END_IF;
   
   	2:(*OPEN RAW WATER OUTLET VALVE, MV201*)
   		(*MV-101 , Raw Water Inlet Valve Control*)
   		_MV_101_SR.EnableIn 	:= 1;
   		_MV_101_SR.Set			:= HMI_LIT101.AL;
   		_MV_101_SR.Reset		:= HMI_LIT101.AH;
   		SETD(_MV_101_SR);
   		_MV101_AutoInp			:= _MV_101_SR.Out;
   
   		_P_RAW_WATER_DUTY_SR.EnableIn	:= 1;
   		_P_RAW_WATER_DUTY_SR.Set		:= HMI_MV201.Status =2 AND HMI_LIT301.AL;
   
   		_P_RAW_WATER_DUTY_SR.Reset		:= HMI_MV201.Status <>2 OR HMI_LIT301.AH;
   		SETD(_P_RAW_WATER_DUTY_SR);
   		_P_RAW_WATER_DUTY_AutoInp	:= _P_RAW_WATER_DUTY_SR.Out;
   
   		IF HMI_P1_SHUTDOWN THEN
   				HMI_P1_STATE	:=3;
   				HMI_P1_SHUTDOWN	:=0;
   		END_IF;
   
   
   
   
   	3:  _MV_101_SR.EnableIn 	:= 1;
   		_MV_101_SR.Set			:= HMI_LIT101.AL;
   		_MV_101_SR.Reset		:= HMI_LIT101.AH;
   		SETD(_MV_101_SR);
   		_MV101_AutoInp			:= _MV_101_SR.Out;
   
   		_P_RAW_WATER_DUTY_SR.EnableIn	:= 1;
   		_P_RAW_WATER_DUTY_SR.Set		:= HMI_MV201.Status =2 AND HMI_LIT301.AL;
   
   		_P_RAW_WATER_DUTY_SR.Reset		:= HMI_MV201.Status <>2 OR HMI_LIT301.AH;
   		SETD(_P_RAW_WATER_DUTY_SR);
   		_P_RAW_WATER_DUTY_AutoInp	:= _P_RAW_WATER_DUTY_SR.Out;
   
   
   		IF  HMI_LIT101.AH AND  HMI_LIT301.AH   THEN
   			_MV101_AutoInp			:= 0;
   			_P_RAW_WATER_DUTY_AutoInp	:= 0;
   			HMI_P1_STATE	:=2;
   		END_IF;
   
   		IF 	HMI_P1_SHUTDOWN THEN
   				HMI_P1_STATE	:=1;
   				HMI_P1_SHUTDOWN	:=0;
   		END_IF;
   
   
   
   
   ELSE
   	HMI_P1_STATE:=1;
   END_CASE;
   
   (*
   
   IF HMI_SHUTDOWN_FLUSHING.ON AND HMI_P5_SD_FLUSHING_DONE.ON THEN
   				HMI_PLANT.STOP	:=1;
   				IF HMI_PLANT.STOP THEN
   					HMI_PLANT.STOP	:=0;
   				END_IF;
   				HMI_SHUTDOWN_FLUSHING.ON :=0;
   
   END_IF;
   *)
END_ROUTINE

ROUTINE MainRoutine   (* ladder *)
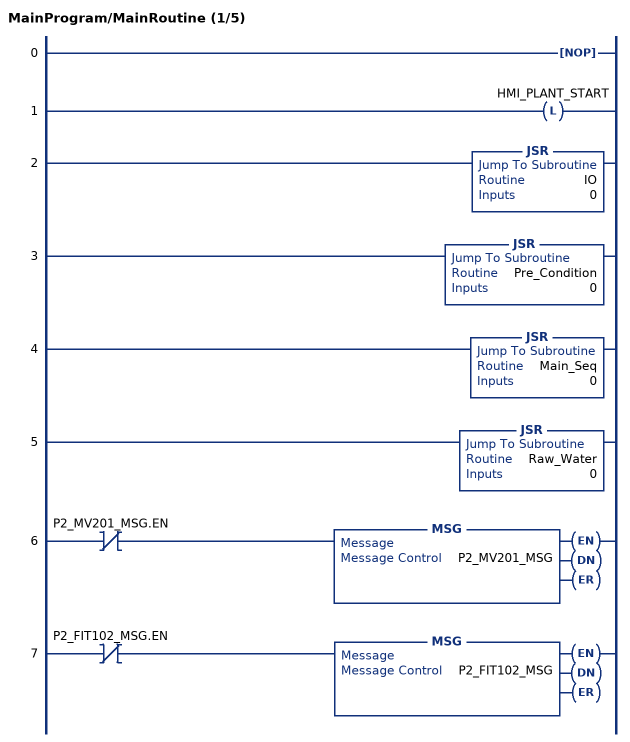
   0: NOP();
   1: OTL(HMI_PLANT_START);
   2: JSR(IO,0);
   3: JSR(Pre_Condition,0);
   4: JSR(Main_Seq,0);
   5: JSR(Raw_Water,0);
   6: XIO(P2_MV201_MSG.EN)MSG(P2_MV201_MSG);
   7: XIO(P2_FIT102_MSG.EN)MSG(P2_FIT102_MSG);
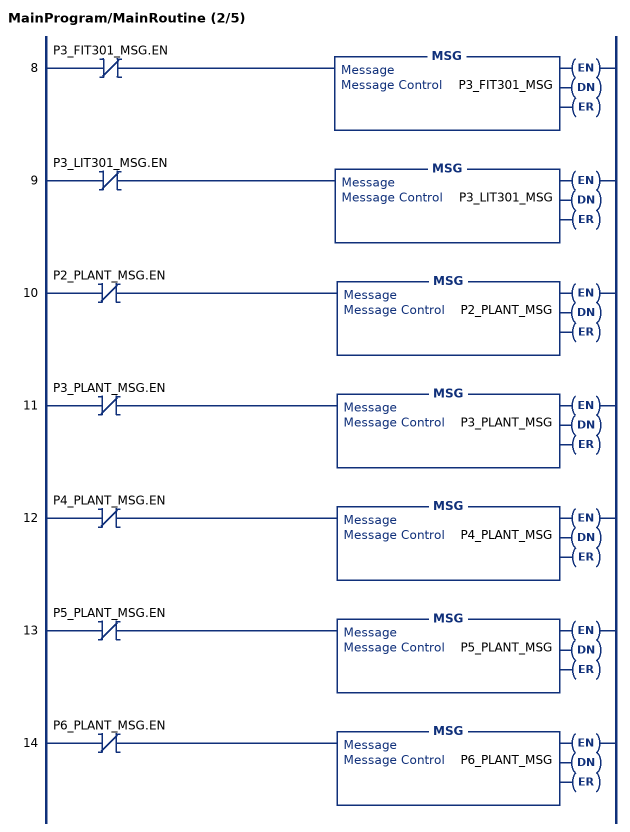
   8: XIO(P3_FIT301_MSG.EN)MSG(P3_FIT301_MSG);
   9: XIO(P3_LIT301_MSG.EN)MSG(P3_LIT301_MSG);
   10: XIO(P2_PLANT_MSG.EN)MSG(P2_PLANT_MSG);
   11: XIO(P3_PLANT_MSG.EN)MSG(P3_PLANT_MSG);
   12: XIO(P4_PLANT_MSG.EN)MSG(P4_PLANT_MSG);
   13: XIO(P5_PLANT_MSG.EN)MSG(P5_PLANT_MSG);
   14: XIO(P6_PLANT_MSG.EN)MSG(P6_PLANT_MSG);
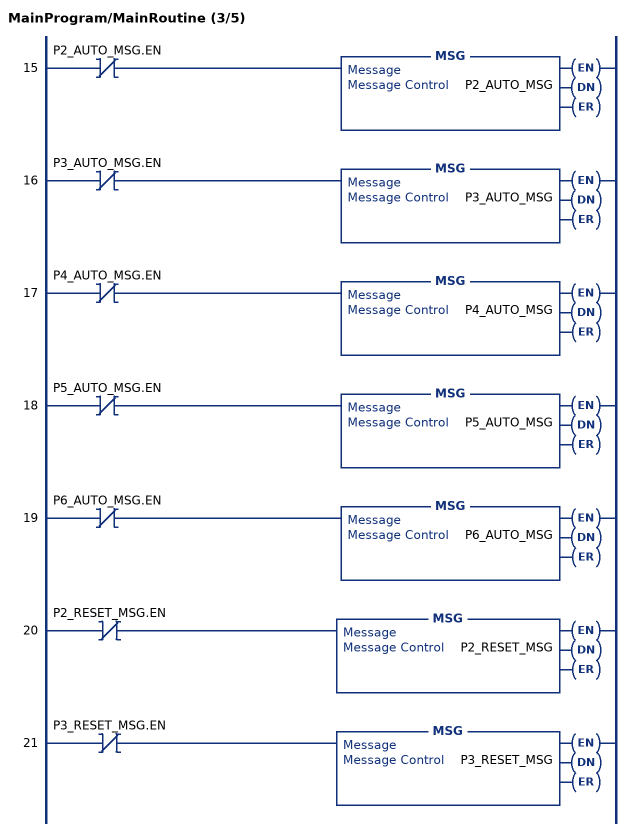
   15: XIO(P2_AUTO_MSG.EN)MSG(P2_AUTO_MSG);
   16: XIO(P3_AUTO_MSG.EN)MSG(P3_AUTO_MSG);
   17: XIO(P4_AUTO_MSG.EN)MSG(P4_AUTO_MSG);
   18: XIO(P5_AUTO_MSG.EN)MSG(P5_AUTO_MSG);
   19: XIO(P6_AUTO_MSG.EN)MSG(P6_AUTO_MSG);
   20: XIO(P2_RESET_MSG.EN)MSG(P2_RESET_MSG);
   21: XIO(P3_RESET_MSG.EN)MSG(P3_RESET_MSG);
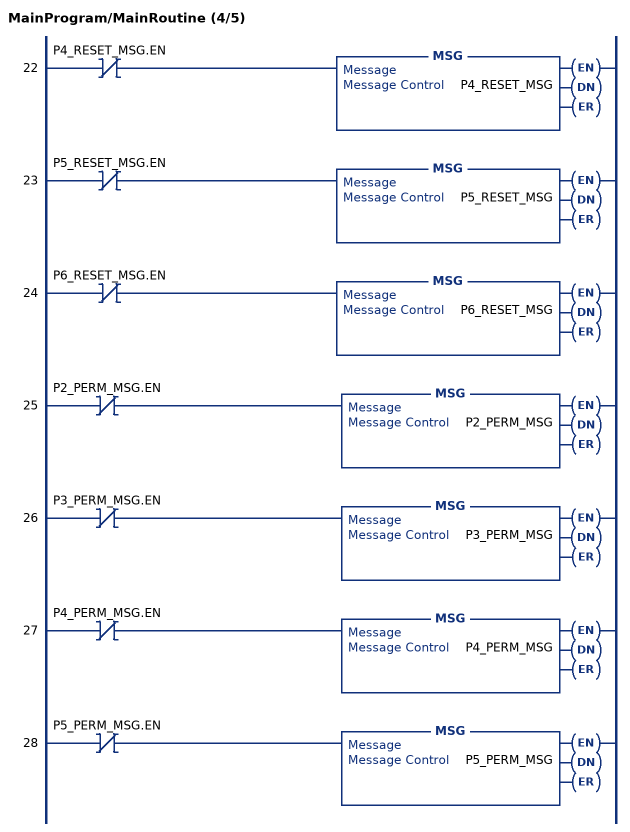
   22: XIO(P4_RESET_MSG.EN)MSG(P4_RESET_MSG);
   23: XIO(P5_RESET_MSG.EN)MSG(P5_RESET_MSG);
   24: XIO(P6_RESET_MSG.EN)MSG(P6_RESET_MSG);
   25: XIO(P2_PERM_MSG.EN)MSG(P2_PERM_MSG);
   26: XIO(P3_PERM_MSG.EN)MSG(P3_PERM_MSG);
   27: XIO(P4_PERM_MSG.EN)MSG(P4_PERM_MSG);
   28: XIO(P5_PERM_MSG.EN)MSG(P5_PERM_MSG);
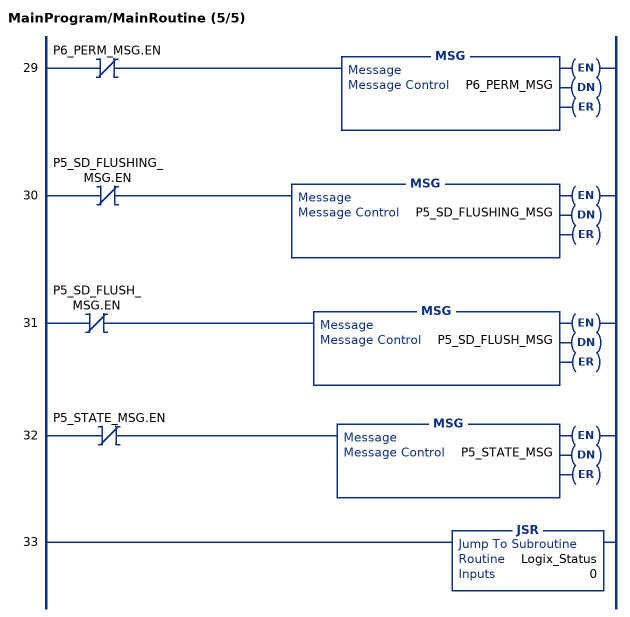
   29: XIO(P6_PERM_MSG.EN)MSG(P6_PERM_MSG);
   30: XIO(P5_SD_FLUSHING_MSG.EN)MSG(P5_SD_FLUSHING_MSG);
   31: XIO(P5_SD_FLUSH_MSG.EN)MSG(P5_SD_FLUSH_MSG);
   32: XIO(P5_STATE_MSG.EN)MSG(P5_STATE_MSG);
   33: JSR(Logix_Status,0);
END_ROUTINE

ROUTINE Pre_Condition   (* structured text *)
      (*RESET ALL INSTRUMENT*)
   IF HMI_PLANT_RESET.ON THEN
   	HMI_MV101.Reset	:=1;
   	HMI_P101.Reset	:=1;
   	HMI_P102.Reset	:=1;
   END_IF;
   
   (*ALL INSTRUMENT IN AUTO MODE*)
   IF HMI_PLANT_AUTO.ON THEN
   	HMI_MV101.Auto	:=1;
   	HMI_P101.Auto	:=1;
   	HMI_P102.Auto	:=1;
   END_IF;
   
   (*ALL INSTRUMENT IN MANUAL MODE*)
   IF HMI_PLANT_AUTO.OFF THEN
   	HMI_MV101.Auto	:=0;
   	HMI_P101.Auto	:=0;
   	HMI_P102.Auto	:=0;
   END_IF;
   
   (*P1 PERMISSIVE*)
   HMI_P1_PERMISSIVE.ON 	:= HMI_MV101.Avl AND (HMI_P101.Avl OR HMI_P102.Avl);
   
   (*PLANT PERMISSIVE*)
   HMI_PLANT_READY 	:= HMI_P1_PERMISSIVE.ON AND HMI_P2_PERMISSIVE.ON AND HMI_P3_PERMISSIVE.ON AND HMI_P4_PERMISSIVE.ON AND HMI_P5_PERMISSIVE.ON AND HMI_P6_PERMISSIVE.ON;
   
   (*Enable Flow Totalising*)
   _FIT101_Tot_Enb 		:= HMI_MV101.status=2;
   
   (*
   TON_FIT102_TM.PRE 			:= 	3*1000;
   TON_FIT102_TM.TimerEnable 	:=  HMI_FIT201.ALL AND HMI_P_RAW_WATER_DUTY.Pump_Running  ;
   TONR(TON_FIT102_TM);
   *)
   
   TON_FIT102_P1_TM.PRE			:= 	10*1000;
   TON_FIT102_P1_TM.TimerEnable 	:=  HMI_FIT201.ALL AND HMI_P101.STATUS=2 ;
   TONR(TON_FIT102_P1_TM);
   
   TON_FIT102_P2_TM.PRE			:= 	10*1000;
   TON_FIT102_P2_TM.TimerEnable 	:=  HMI_FIT201.ALL AND HMI_P102.STATUS=2 ;
   TONR(TON_FIT102_P2_TM);
   
   
   (*-------------------------------------------------------------------------------------------------------------*)
   (*P101 Permissive*)
   HMI_P101.Permissive.0 	:= HMI_LIT101.HTY AND NOT HMI_LIT101.ALL;;
   HMI_P101.Permissive.1 	:= HMI_MV201.Status=2; (*Status from P2*)
   HMI_P101.Permissive.2 	:= 1;
   HMI_P101.Permissive.3 	:= 1;
   HMI_P101.Permissive.4 	:= 1;
   HMI_P101.Permissive.5 	:= 1;
   HMI_P101.Permissive.6 	:= 1;
   HMI_P101.Permissive.7 	:= 1;
   HMI_P101.Permissive.8 	:= 1;
   HMI_P101.Permissive.9 	:= 1;
   HMI_P101.Permissive.10 	:= 1;
   HMI_P101.Permissive.11 	:= 1;
   HMI_P101.Permissive.12 	:= 1;
   HMI_P101.Permissive.13	:= 1;
   HMI_P101.Permissive.14	:= 1;
   HMI_P101.Permissive.15 	:= 1;
   
   HMI_P101_MSG.PERMISSIVE1 := HMI_P101.Permissive.0;
   HMI_P101_MSG.PERMISSIVE2 := HMI_P101.Permissive.1;
   HMI_P101_MSG.PERMISSIVE3 := 0;
   HMI_P101_MSG.PERMISSIVE4 := 0;
   HMI_P101_MSG.PERMISSIVE5 := 0;
   
   (*P102 Permissive*)
   HMI_P102.Permissive.0 	:= HMI_LIT101.HTY AND NOT HMI_LIT101.ALL;;
   HMI_P102.Permissive.1 	:= HMI_MV201.Status=2; (*Status from P2*)
   HMI_P102.Permissive.2 	:= 1;
   HMI_P102.Permissive.3 	:= 1;
   HMI_P102.Permissive.4 	:= 1;
   HMI_P102.Permissive.5 	:= 1;
   HMI_P102.Permissive.6 	:= 1;
   HMI_P102.Permissive.7 	:= 1;
   HMI_P102.Permissive.8 	:= 1;
   HMI_P102.Permissive.9 	:= 1;
   HMI_P102.Permissive.10 	:= 1;
   HMI_P102.Permissive.11 	:= 1;
   HMI_P102.Permissive.12 	:= 1;
   HMI_P102.Permissive.13	:= 1;
   HMI_P102.Permissive.14	:= 1;
   HMI_P102.Permissive.15 	:= 1;
   
   HMI_P102_MSG.PERMISSIVE1 := HMI_P102.Permissive.0;
   HMI_P102_MSG.PERMISSIVE2 := HMI_P102.Permissive.1;
   HMI_P102_MSG.PERMISSIVE3 := 0;
   HMI_P102_MSG.PERMISSIVE4 := 0;
   HMI_P102_MSG.PERMISSIVE5 := 0;
   
   (*------------------------------------------------------------------------------*)
   (*P101 Shutdown*)
   HMI_P101.SD.0 	:= HMI_LIT101.HTY AND HMI_LIT101.ALL;
   HMI_P101.SD.1 	:= HMI_P101.STATUS=2 AND HMI_MV201.Status<>2; (*Status from P2*)
   HMI_P101.SD.2 	:= TON_FIT102_P1_TM.DN;
   HMI_P101.SD.3 	:= 0;
   HMI_P101.SD.4 	:= 0;
   HMI_P101.SD.5 	:= 0;
   HMI_P101.SD.6 	:= 0;
   HMI_P101.SD.7 	:= 0;
   HMI_P101.SD.8 	:= 0;
   HMI_P101.SD.9 	:= 0;
   HMI_P101.SD.10 	:= 0;
   HMI_P101.SD.11 	:= 0;
   HMI_P101.SD.12 	:= 0;
   HMI_P101.SD.13 	:= 0;
   HMI_P101.SD.14 	:= 0;
   HMI_P101.SD.15 	:= 0;
   
   HMI_P101_MSG.SHUTODWN1 := HMI_P101.Shutdown.0;
   HMI_P101_MSG.SHUTODWN2 := HMI_P101.Shutdown.1;
   HMI_P101_MSG.SHUTODWN3 := HMI_P101.Shutdown.2;
   HMI_P101_MSG.SHUTODWN4 := 0;
   HMI_P101_MSG.SHUTODWN5 := 0;
   
   (*P102 Shutdown*)
   HMI_P102.SD.0 	:= HMI_LIT101.HTY AND HMI_LIT101.ALL;
   HMI_P102.SD.1 	:= HMI_P102.STATUS=2 AND HMI_MV201.Status<>2; (*Status from P2*)
   HMI_P102.SD.2 	:= TON_FIT102_P2_TM.DN;
   HMI_P102.SD.3 	:= 0;
   HMI_P102.SD.4 	:= 0;
   HMI_P102.SD.5 	:= 0;
   HMI_P102.SD.6 	:= 0;
   HMI_P102.SD.7 	:= 0;
   HMI_P102.SD.8 	:= 0;
   HMI_P102.SD.9 	:= 0;
   HMI_P102.SD.10 	:= 0;
   HMI_P102.SD.11 	:= 0;
   HMI_P102.SD.12 	:= 0;
   HMI_P102.SD.13 	:= 0;
   HMI_P102.SD.14 	:= 0;
   HMI_P102.SD.15 	:= 0;
   
   HMI_P102_MSG.SHUTODWN1 := HMI_P102.Shutdown.0;
   HMI_P102_MSG.SHUTODWN2 := HMI_P102.Shutdown.1;
   HMI_P102_MSG.SHUTODWN3 := HMI_P102.Shutdown.2;
   HMI_P102_MSG.SHUTODWN4 := 0;
   HMI_P102_MSG.SHUTODWN5 := 0;
   
   
   
   
   
END_ROUTINE

ROUTINE Raw_Water   (* function block diagram *)
   SHEET 1
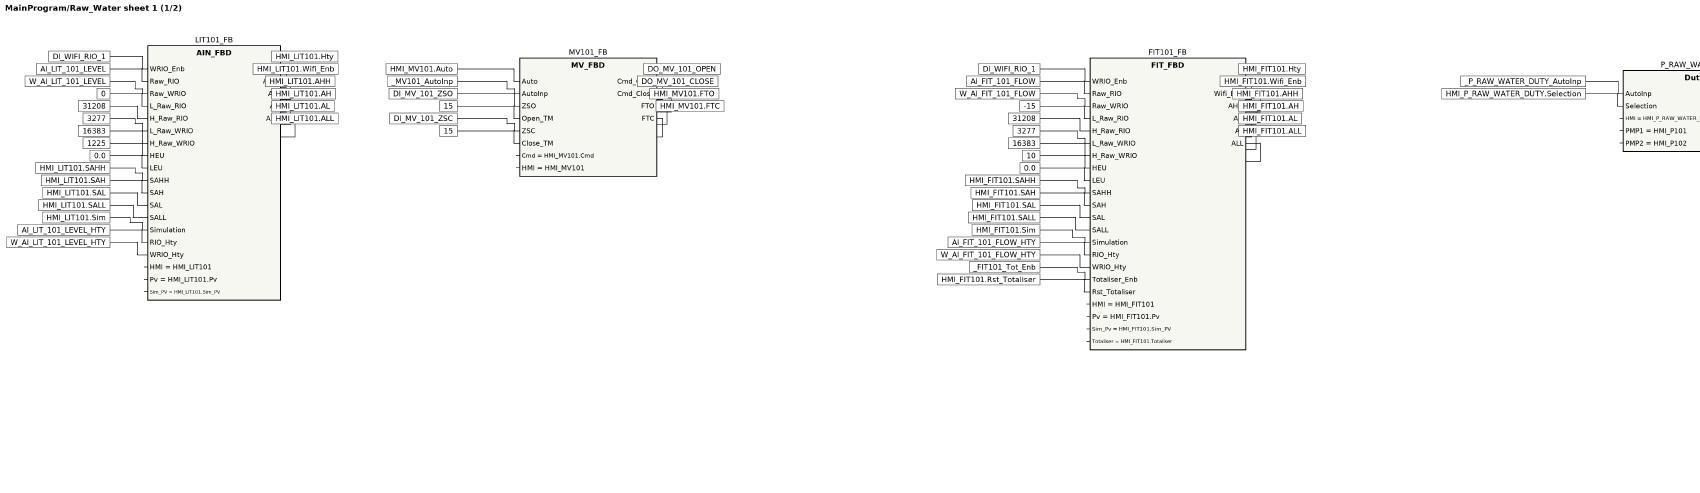
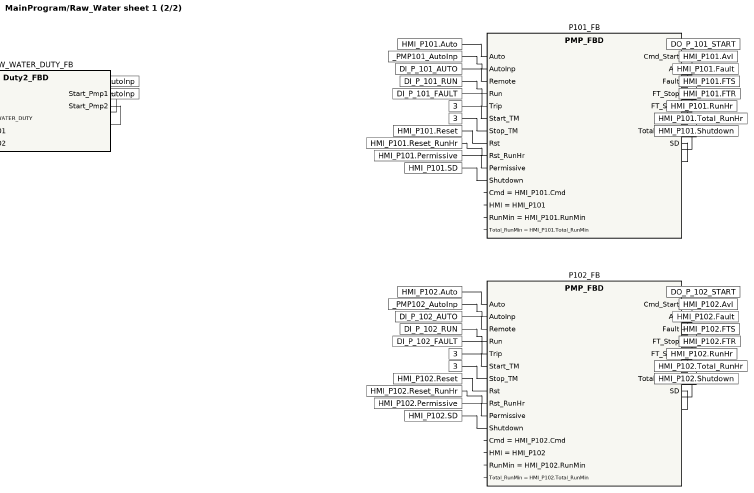
   LIT101_FB : AIN_FBD(WRIO_Enb := DI_WIFI_RIO_1, Raw_RIO := AI_LIT_101_LEVEL, Raw_WRIO := W_AI_LIT_101_LEVEL, L_Raw_RIO := 0, H_Raw_RIO := 31208, L_Raw_WRIO := 3277, H_Raw_WRIO := 16383, HEU := 1225, LEU := 0.0, SAHH := HMI_LIT101.SAHH, SAH := HMI_LIT101.SAH, SAL := HMI_LIT101.SAL, SALL := HMI_LIT101.SALL, Simulation := HMI_LIT101.Sim, RIO_Hty := AI_LIT_101_LEVEL_HTY, WRIO_Hty := W_AI_LIT_101_LEVEL_HTY, HMI := HMI_LIT101, Pv := HMI_LIT101.Pv, Sim_PV := HMI_LIT101.Sim_PV);
   // unwired output reference HMI_LIT101.Wifi_Enb
   HMI_LIT101.AHH := LIT101_FB.AHH;
   HMI_LIT101.Hty := LIT101_FB.Hty;
   HMI_LIT101.AH := LIT101_FB.AH;
   HMI_LIT101.AL := LIT101_FB.AL;
   HMI_LIT101.ALL := LIT101_FB.ALL;
   MV101_FB : MV_FBD(Auto := HMI_MV101.Auto, AutoInp := _MV101_AutoInp, ZSO := DI_MV_101_ZSO, Open_TM := 15, ZSC := DI_MV_101_ZSC, Close_TM := 15, Cmd := HMI_MV101.Cmd, HMI := HMI_MV101);
   DO_MV_101_CLOSE := MV101_FB.Cmd_Close;
   DO_MV_101_OPEN := MV101_FB.Cmd_Open;
   HMI_MV101.FTO := MV101_FB.FTO;
   HMI_MV101.FTC := MV101_FB.FTC;
   FIT101_FB : FIT_FBD(WRIO_Enb := DI_WIFI_RIO_1, Raw_RIO := AI_FIT_101_FLOW, Raw_WRIO := W_AI_FIT_101_FLOW, L_Raw_RIO := -15, H_Raw_RIO := 31208, L_Raw_WRIO := 3277, H_Raw_WRIO := 16383, HEU := 10, LEU := 0.0, SAHH := HMI_FIT101.SAHH, SAH := HMI_FIT101.SAH, SAL := HMI_FIT101.SAL, SALL := HMI_FIT101.SALL, Simulation := HMI_FIT101.Sim, RIO_Hty := AI_FIT_101_FLOW_HTY, WRIO_Hty := W_AI_FIT_101_FLOW_HTY, Totaliser_Enb := _FIT101_Tot_Enb, Rst_Totaliser := HMI_FIT101.Rst_Totaliser, HMI := HMI_FIT101, Pv := HMI_FIT101.Pv, Sim_Pv := HMI_FIT101.Sim_PV, Totaliser := HMI_FIT101.Totaliser);
   HMI_FIT101.Wifi_Enb := FIT101_FB.Wifi_Enb;
   HMI_FIT101.AHH := FIT101_FB.AHH;
   HMI_FIT101.Hty := FIT101_FB.Hty;
   HMI_FIT101.AH := FIT101_FB.AH;
   HMI_FIT101.AL := FIT101_FB.AL;
   HMI_FIT101.ALL := FIT101_FB.ALL;
   P_RAW_WATER_DUTY_FB : Duty2_FBD(AutoInp := _P_RAW_WATER_DUTY_AutoInp, Selection := HMI_P_RAW_WATER_DUTY.Selection, HMI := HMI_P_RAW_WATER_DUTY, PMP1 := HMI_P101, PMP2 := HMI_P102);
   _PMP101_AutoInp := P_RAW_WATER_DUTY_FB.Start_Pmp1;
   _PMP102_AutoInp := P_RAW_WATER_DUTY_FB.Start_Pmp2;
   P101_FB : PMP_FBD(Auto := HMI_P101.Auto, AutoInp := _PMP101_AutoInp, Remote := DI_P_101_AUTO, Run := DI_P_101_RUN, Trip := DI_P_101_FAULT, Start_TM := 3, Stop_TM := 3, Rst := HMI_P101.Reset, Rst_RunHr := HMI_P101.Reset_RunHr, Permissive := HMI_P101.Permissive, Shutdown := HMI_P101.SD, Cmd := HMI_P101.Cmd, HMI := HMI_P101, RunMin := HMI_P101.RunMin, Total_RunMin := HMI_P101.Total_RunMin);
   P102_FB : PMP_FBD(Auto := HMI_P102.Auto, AutoInp := _PMP102_AutoInp, Remote := DI_P_102_AUTO, Run := DI_P_102_RUN, Trip := DI_P_102_FAULT, Start_TM := 3, Stop_TM := 3, Rst := HMI_P102.Reset, Rst_RunHr := HMI_P102.Reset_RunHr, Permissive := HMI_P102.Permissive, Shutdown := HMI_P102.SD, Cmd := HMI_P102.Cmd, HMI := HMI_P102, RunMin := HMI_P102.RunMin, Total_RunMin := HMI_P102.Total_RunMin);
   HMI_P101.Total_RunHr := P101_FB.Total_RunHr;
   HMI_P101.Shutdown := P101_FB.SD;
   HMI_P102.Total_RunHr := P102_FB.Total_RunHr;
   HMI_P102.Shutdown := P102_FB.SD;
   DO_P_101_START := P101_FB.Cmd_Start;
   HMI_P101.RunHr := P101_FB.RunHr;
   DO_P_102_START := P102_FB.Cmd_Start;
   HMI_P102.RunHr := P102_FB.RunHr;
   HMI_P101.Fault := P101_FB.Fault;
   HMI_P102.Fault := P102_FB.Fault;
   HMI_P101.Avl := P101_FB.Avl;
   HMI_P101.FTS := P101_FB.FT_Stop;
   HMI_P101.FTR := P101_FB.FT_Start;
   HMI_P102.Avl := P102_FB.Avl;
   HMI_P102.FTS := P102_FB.FT_Stop;
   HMI_P102.FTR := P102_FB.FT_Start;
END_ROUTINE
END_PROGRAM
